(* revision histroy
hm	18. jun. 2008	rev 1.0
	original release

hm	20. sep. 2008	rev 1.1
	changed length of input string from 20 to 12
*)	
END_FUNCTION

(* POU String/BIN_TO_BYTE, ST *)
FUNCTION BIN_TO_BYTE : BYTE
VAR_INPUT
	BIN : STRING(12);
END_VAR
VAR
	pt : POINTER TO BYTE;
	i: INT;
	X: BYTE;
	stop: INT;
END_VAR

(*
version 1.1	20. sep. 2008
programmer 	hugo
tested by	oscat

BINARY_TO_byte converts a binary string into a byte.

*)
pt := ADR(bin);
stop := LEN(bin);
FOR I := 1 TO stop DO
	(* read the first character and subtract 48 to get value in decimal 0 = 48 *)
	x := pt^;
	(* calculate the value of the digit *)
	IF X = 48 OR X = 49 THEN
		BIN_TO_BYTE := SHL(BIN_TO_BYTE,1) + X - 48;
	END_IF;
	pt := pt + 1;
END_FOR;



(* revision histroy
hm	18. jun. 2008	rev 1.0
	original release

hm	20. sep. 2008	rev 1.1
	changed length of input string from 20 to 12

*)	
END_FUNCTION

(* POU String/OCT_TO_BYTE, ST *)
FUNCTION OCT_TO_BYTE : BYTE
VAR_INPUT
	OCT : STRING(10);
END_VAR
VAR
	pt : POINTER TO BYTE;
	i: INT;
	X: BYTE;
	stop: INT;
END_VAR

(*
version 1.1	20. sep. 2008
programmer 	hugo
tested by		oscat

OCT_TO_BYTE converts a octagonal string into a byte.

*)
pt := ADR(oct);
stop := LEN(oct);
FOR I := 1 TO stop DO
	(* read the first character and subtract 48 to get value in decimal 0 = 48 *)
	x := pt^;
	(* calculate the value of the digit *)
	IF X > 47 AND x < 56 THEN
		OCT_TO_BYTE := SHL(OCT_TO_BYTE,3) + X - 48;
	END_IF;
	pt := pt + 1;
END_FOR;



(* revision histroy
hm	18. jun. 2008	rev 1.0
	original release

hm	20. sep. 2008	rev 1.1
	changed length of input string from 20 to 10

*)	
END_FUNCTION

(* POU String/HEX_TO_BYTE, ST *)
FUNCTION HEX_TO_BYTE : BYTE
VAR_INPUT
	HEX : STRING(5);
END_VAR
VAR
	pt : POINTER TO BYTE;
	i: INT;
	X: BYTE;
	stop: INT;
END_VAR

(*
version 1.1	20. sep. 2008
programmer 	hugo
tested by		oscat

HEX_TO_BYTE converts a Hexadecimal string into a byte.

*)
pt := ADR(hex);
stop := LEN(hex);
FOR I := 1 TO stop DO
	(* read the first character and subtract 48 to get value in decimal 0 = 48 *)
	x := pt^;
	(* calculate the value of the digit *)
	IF X > 47 AND x < 58 THEN
		HEX_TO_BYTE := SHL(HEX_TO_BYTE,4) + X - 48;
	ELSIF X > 64 AND X < 71 THEN
		HEX_TO_BYTE := SHL(HEX_TO_BYTE,4) + X - 55;
	ELSIF X > 96 AND X < 103 THEN
		HEX_TO_BYTE := SHL(HEX_TO_BYTE,4) + X - 87;
	END_IF;
	pt := pt + 1;
END_FOR;




(* revision histroy
hm	18. jun. 2008	rev 1.0
	original release

hm	20. sep.2008	rev 1.1
	changed length of input string from 20 to 5

*)	
END_FUNCTION

(* POU String/DEC_TO_BYTE, ST *)
FUNCTION DEC_TO_BYTE : BYTE
VAR_INPUT
	DEC : STRING(10);
END_VAR
VAR
	pt : POINTER TO BYTE;
	i: INT;
	X: BYTE;
	stop: INT;
END_VAR

(*
version 1.1	30. sep 2008
programmer 	hugo
tested by		oscat

DEC_TO_byte converts a decimal string into a byte.

*)
pt := ADR(dec);
stop := LEN(DEC);
FOR I := 1 TO stop DO
	(* read the first character and subtract 48 to get value in decimal 0 = 48 *)
	x := pt^;
	(* calculate the value of the digit *)
	IF X > 47 AND x < 58 THEN
		DEC_TO_BYTE := DEC_TO_BYTE * 10 + X - 48;
	END_IF;
	pt := pt + 1;
END_FOR;



(* revision histroy
hm	20. jun. 2008	rev 1.0
	original release

hm	30. sep.2008	rev 1.1
	changed length of input string from 20 to 10
	corrected an error where decoding of characters 8 and 9 would fail

*)	
END_FUNCTION

(* POU String/CLEAN, ST *)
FUNCTION CLEAN : STRING(STRING_LENGTH)
VAR_INPUT
	IN : STRING(STRING_LENGTH);
	CX : STRING(80);
END_VAR
VAR
	pos: INT := 1;
	stop: INT;
END_VAR


(*
version 1.0	18. jun. 2008
programmer 	hugo
tested by	oscat

Clean deletes all characters from a string except the ones specified in CX.

*)
(* copy input string *)
CLEAN := IN;
stop := LEN(in);
WHILE pos <= stop DO
	IF FIND(cx, MID(CLEAN, 1, pos)) > 0 THEN
		(* charcter found skip to next one *)
		pos := pos + 1;
	ELSE
		(* wrong chracter needs to be deleted *)
		CLEAN := DELETE(CLEAN, 1, pos);
		stop := stop - 1;	(* the string is one character shorter now *)
	END_IF;
END_WHILE;



(* revision history

hm		18. jun. 2008	rev 1.0		
	original version 


*)
END_FUNCTION

(* POU String/IS_CC, ST *)
FUNCTION IS_CC : BOOL
VAR_INPUT
	str : STRING(STRING_LENGTH);
	cmp : STRING(STRING_LENGTH);
END_VAR
VAR
	L: INT;
	pos: INT;
END_VAR

(*
version 1.1	29. mar. 2008
programmer 	Tobias
tested by	hugo

ISC_CC testet ob ein string nur aus Zeichen des Strings CMP besteht.

*)
L := LEN(str);
FOR pos := 1 TO L DO
	IF FIND(CMP,MID(str,1,pos)) = 0 THEN RETURN; END_IF;
END_FOR;
IS_CC := L > 0;



(* revision history
hm	19. mar 2008	rev 1.0
	original version

hm	29. mar. 2008	rev 1.1
	changed STRING to STRING(STRING_LENGTH)
*)
END_FUNCTION

(* POU Mathematical/CMP, ST *)
FUNCTION CMP : BOOL
VAR_INPUT
	X,Y : REAL;
	N : INT;
END_VAR
VAR
	tmp : REAL;
END_VAR


(*
	version 1.0	12 mar 2008
	programmer 	hugo
	tested by		tobias

this function checks two inputs x and y if they are identical with the first N digits
example : cmp(3.141516,3.141517,6 is true.

*)
tmp := ABS(x);
IF tmp > 0 THEN
	tmp := EXP10(FLOOR(LOG(tmp))-N+1);
ELSE
	tmp := EXP10(tmp);
END_IF;
CMP := ABS(X - Y) < tmp;


(* revision history
hm	12. mar. 2008	rev 1.0
	original version

*)
END_FUNCTION

(* POU Mathematical/EXP10, ST *)
FUNCTION EXP10 : REAL
VAR_INPUT
	X : REAL;
END_VAR
VAR
END_VAR

(*
version 1.0	 2 dec 2007
programmer 	hugo
tested by		tobias

this function calculates the exponent to the basis 10
exp10(3) = 1000

*)
EXP10 := EXP(X * 2.30258509299405);

(* revision history
hm	2. dec 2007		rev 1.0
	original version

*)
END_FUNCTION

(* POU String/FSTRING_TO_WEEK, ST *)
FUNCTION FSTRING_TO_WEEK : BYTE
VAR_INPUT
	WEEK : STRING(60);
	LANG : INT;
END_VAR
VAR
	pos: INT;
END_VAR


(*
version 1.1	25. oct. 2008
programmer 	hugo
tested by	oscat

FSTRING_TO_WEEK converts a list of weekdays into a byte where each bit represents a day of the week.
bit 6 = mo, 0 = su;

*)
pos := FIND(WEEK, ',');
WHILE pos > 0 DO
	FSTRING_TO_WEEK := FSTRING_TO_WEEK OR SHR(BYTE#128, FSTRING_TO_WEEKDAY(MID(WEEK, pos - 1, 1), LANG));
	WEEK := RIGHT(WEEK, LEN(Week) - pos);
	pos := FIND(WEEK, ',');
END_WHILE;
FSTRING_TO_WEEK := (FSTRING_TO_WEEK OR SHR(BYTE#128, FSTRING_TO_WEEKDAY(WEEK, LANG))) AND BYTE#127;


(* revision histroy
hm	18. jun. 2008	rev 1.0
	original release

hm	25. oct. 2008	rev 1.1
	using language defauls and input lang
*)	
END_FUNCTION

(* POU String/FSTRING_TO_WEEKDAY, ST *)
FUNCTION FSTRING_TO_WEEKDAY : INT
VAR_INPUT
	WDAY : STRING(20);
	LANG : INT;
END_VAR
VAR
	tmp: STRING(2);
	i: INT;
	ly: INT;
END_VAR


(*
version 1.2	25. oct. 2008
programmer 	hugo
tested by	oscat

FSTRING_TO_WEEKDAY converts a weekday string into an integer 1..7.

*)
IF LANG = 0 THEN ly := LANGUAGE.DEFAULT; ELSE ly := MIN(LANG, LANGUAGE.LMAX); END_IF;
(* tmp needs to be calculated first otherwise find can return wrong values *)
tmp := TRIM(wday);
tmp := CAPITALIZE(LOWERCASE(tmp));
FOR i := 1 TO 7 DO
	IF language.WEEKDAYS2[ly, i] = tmp THEN
		FSTRING_TO_WEEKDAY := i;
		RETURN;
	END_IF;
END_FOR
FSTRING_TO_WEEKDAY := STRING_TO_INT(WDAY);




(* revision histroy
hm	18. jun. 2008	rev 1.0
	original release

hm	18. jul. 2008	rev 1.1
	changed nested call of left(trim()) for compatibility reasons

hm	25. oct. 2008	rev 1.2
	using language constants
*)	
END_FUNCTION

(* POU String/TRIM, ST *)
FUNCTION TRIM : STRING(STRING_LENGTH)
VAR_INPUT
	str : STRING(STRING_LENGTH);
END_VAR
VAR
	pos: INT;
END_VAR

(*
version 1.2	29. mar. 2008
programmer 	hugo
tested by	tobias

the function deletes all blanks within a string.

*)
TRIM := str;
REPEAT
	pos := FIND(trim,' ');
	IF pos > 0 THEN TRIM := REPLACE(TRIM,'',1,pos); END_IF;
UNTIL pos = 0	END_REPEAT;


(* revision histroy
hm	6.10.2006		rev 1.0
	original release

hm	20. mar. 2008	rev 1.1
	avoid to call replace with pos = 0 because some systems will produce an error

hm	29. mar. 2008	rev 1.2
	changed STRING to STRING(STRING_LENGTH)
*)
END_FUNCTION

(* POU String/CAPITALIZE, ST *)
FUNCTION CAPITALIZE : STRING(STRING_LENGTH)
VAR_INPUT
	str : STRING(STRING_LENGTH);
END_VAR
VAR
	PT : POINTER TO BYTE;
	pos : INT;
	L : INT;
	first : BOOL := TRUE;
END_VAR

(*
version 1.2	20. jun. 2008
programmer 	hugo
tested by		tobias

capitalize returns str with all first letters after a blank or beginning of the string are converted to uppercase.

*)
PT := ADR(CAPITALIZE);
CAPITALIZE := str;
L := LEN(str);
FOR pos := 1 TO l DO
	IF first THEN pt^ := TO_UPPER(pt^);	END_IF;
	(* remember in first if the next char needs to capitalized *)
	first := pt^= 32;
	PT := pt + 1;
END_FOR;

(* revision histroy
hm		4. mar 2008	rev 1.0
	original release

hm	29. mar. 2008	rev 1.1
	changed STRING to STRING(STRING_LENGTH)

hm	20. jun. 2008	rev 1.2
	improved performance

*)	
END_FUNCTION

(* POU String/TO_UPPER, ST *)
FUNCTION TO_UPPER : BYTE
VAR_INPUT
	IN : BYTE;
END_VAR
VAR
END_VAR

(*
version 1.3	16. jan. 2009
programmer 	hugo
tested by		oscat

to_upper converts a character from lowercase to uppercase

*)
IF in > 96 AND in < 123 THEN
   TO_UPPER := in AND 16#DF;
ELSIF in > 223 AND in <> 247 AND in <> 255 AND setup.EXTENDED_ASCII THEN
   TO_UPPER := in AND 16#DF;
ELSE
   TO_UPPER := in;
END_IF;




(* revision history
hm	6. mar. 2008	rev 1.0
	original version

hm	19. oct. 2008	rev 1.1
	changed setup constants

ks	25. oct. 2008	rev 1.2
	optimized code

hm 16. jan 2009	rev 1.3
	corrected an error in module

*)
END_FUNCTION

(* POU String/LOWERCASE, ST *)
FUNCTION LOWERCASE : STRING(STRING_LENGTH)
VAR_INPUT
	str : STRING(STRING_LENGTH);
END_VAR
VAR
	PT : POINTER TO BYTE;
	pos: INT;
	l: INT;
END_VAR

(*
version 1.3	29. mar. 2008
programmer 	hugo
tested by		tobias

lowercase returns str while all letters A..Z and Ä.Ö,Ü are converted to lowercase.

*)
PT := ADR(LOWERCASE);
lowercase := str;
l := LEN(str);
FOR pos := 1 TO l DO
	pt^ := TO_LOWER(pt^);
	PT := PT + 1;
END_FOR;

(* revision histroy
hm	6. oct. 2006	rev 1.0
	original release

hm	4. feb. 2008	rev 1.1
	improved performance
	added Ä.Ö,Ü

hm	6. mar. 2008	rev 1.2
	added support for exteded Ascii

hm	29. mar. 2008	rev 1.3
	changed STRING to STRING(STRING_LENGTH)
*)	
END_FUNCTION

(* POU String/TO_LOWER, ST *)
FUNCTION TO_LOWER : BYTE
VAR_INPUT
	IN : BYTE;
END_VAR
VAR
END_VAR

(*
version 1.2	25. oct 2008
programmer 	hugo
tested by		tobias

to_lower converts a character from uppercase to lowercase

*)
IF in > 64 AND in < 91 THEN
   TO_LOWER := in OR 16#20;
ELSIF (in > 191 AND in < 223) AND in <> 215 AND setup.EXTENDED_ASCII THEN
   TO_LOWER := in OR 16#20;
ELSE
   TO_LOWER := in;
END_IF;


(* revision history
hm	6. mar. 2008	rev 1.0
	original version

hm	19. oct. 2008	rev 1.1
	changed setup constants

ks	25. oct. 2008	rev 1.2
	optimized code
*)
END_FUNCTION

(* POU Building/electrical/TIMER_EXT, ST *)
FUNCTION_BLOCK TIMER_EXT
VAR_INPUT
	ENA : BOOL := TRUE;
	ON : BOOL;
	OFF : BOOL;
	MAN : BOOL;
	SWITCH : BOOL;
	DT_IN : DT;
	SUN_RISE : TOD;
	SUN_SET : TOD;
	HOLIDAY : BOOL;
END_VAR
VAR_INPUT CONSTANT
	T_DEBOUNCE : TIME := T#100ms;
	T_RISE_START : TIME;
	T_RISE_STOP : TIME;
	T_SET_START : TIME;
	T_SET_STOP : TIME;
	T_DAY_START : TOD;
	T_DAY_STOP : TOD;
	ENABLE_SATURDAY : BOOL;
	ENABLE_SUNDAY : BOOL;
	ENABLE_HOLIDAY : BOOL;
END_VAR
VAR_OUTPUT
	Q : BOOL;
	STATUS: BYTE;
END_VAR
VAR
	mx : MANUAL_2;
	deb : DEBOUNCE;
	tdx: TOD;
	wdx: INT;
	tc : TIME;
	tx: DWORD;
	tl: DWORD;
	qx: BOOL;
	init: BOOL;
END_VAR

(*
version 1.1	6. nov. 2008
programmer 	oscat
tested by	tobias

TIMER_EXT is a twilight timer.
the timer can be programmed to switch lights or other equippment or during twilight times.
in addition to the automatik mode the timer can be stopped and started by a switch at any given time.
An enable input ENA can be used for external control.
two inputs ON and OFF can be used to statically control the output.
the timer can be programmed to work on saturdays, sundays and holidays if required.

*)
(* lösche die millisekunden bei sunrise und sunset *)
SUN_RISE := DWORD_TO_TOD(TOD_TO_DWORD(SUN_RISE) / 1000 * 1000);
SUN_SET := DWORD_TO_TOD(TOD_TO_DWORD(SUN_SET) / 1000 * 1000);

(* measure cycle time tc and make sure this circuitry is not called more then once in 200ms*)
tx := T_PLC_MS();
IF NOT init THEN
	init := TRUE;
	tl := tx;
END_IF;
tc := DWORD_TO_TIME(tx - tl);
IF tc < t#200ms THEN RETURN; END_IF;
tl := tx;

(* debounce *)
deb(in := SWITCH, TD := T_DEBOUNCE, PM := TRUE);

(* read time of day and strip off all milliseconds *)
tdx := DT_TO_TOD(dt_in);
wdx := DAY_OF_WEEK(DT_TO_DATE(dt_in));

(* automatic output control *)
IF deb.Q THEN
	qx := NOT qx;
	status := 110;
ELSIF holiday AND NOT enable_holiday THEN
	qx := FALSE;
ELSIF wdx = 6 AND NOT enable_saturday THEN
	qx := FALSE;
ELSIF wdx = 7 AND NOT enable_sunday THEN
	qx := FALSE;
ELSIF T_day_start > TOD#00:00 AND tdx - T_DAY_START <= tc THEN
	(* turn on at specified daytime *)
	qx := TRUE;
	status := 111;
ELSIF T_DAY_STOP > TOD#00:00 AND tdx - T_DAY_STOP <= tc THEN
	(* turn off at specific daytime *)
	qx := FALSE;
	status := 112;
ELSIF T_RISE_START > T#0s AND tdx - SUN_RISE + T_RISE_START <= tc THEN
	(* turn on before sunrise *)
	qx := TRUE;
	status := 113;
ELSIF T_RISE_STOP > T#0s AND tdx - SUN_RISE - T_RISE_STOP <= tc THEN
	(* turn off after sunrise *)
	qx := FALSE;
	status := 114;
ELSIF T_SET_start > T#0s AND tdx - SUN_SET + T_SET_START <= tc THEN
	(* turn on before sunset *)
	qx := TRUE;
	status := 115;
ELSIF T_SET_STOP > t#0s AND tdx - SUN_SET - T_SET_STOP <= tc THEN
	(* turn off after sunset *)
	qx := FALSE;
	status := 116;
END_IF;


(* mnaual and output control *)
mx(in := qx, ena := ENA, on := ON, off := OFF, man := MAN);
Q := mx.Q;

(* set the status output *)
IF mx.STATUS > 100 THEN status := mx.STATUS; END_IF;



(*
hm 	7. oct. 2008	rev 1.0
	original version

hm	6. nov. 2008	rev 1.1
	added default = true for ena input
*)
END_FUNCTION_BLOCK

(* POU Engineering/automation/MANUAL_2, ST *)
FUNCTION_BLOCK MANUAL_2
VAR_INPUT
	IN : BOOL;
	ENA : BOOL;
	ON : BOOL;
	OFF : BOOL;
	MAN : BOOL;
END_VAR
VAR_OUTPUT
	Q : BOOL;
	STATUS : BYTE;
END_VAR
VAR
END_VAR

(*
version 1.0	22. sep. 2008
programmer 	hugo
tested by	oscat

MANUAL_2 is a manual override for boolean signals.
it has static force high and low as well as a manual input.

*)
IF ena THEN
	IF NOT ON AND NOT OFF THEN
		Q := IN;
		STATUS := 100;
	ELSIF on AND NOT off THEN
		Q := TRUE;
		STATUS := 101;
	ELSIF NOT on AND off THEN
		q := FALSE;
		STATUS := 102;
	ELSE
		Q := MAN;
		STATUS := 103;
	END_IF;
ELSE
	Q := FALSE;
	STATUS := 104;
END_IF;



(* revision history
hm	22. sep. 2008		rev 1.0
	original version

*)
END_FUNCTION_BLOCK

(* POU Building/electrical/TIMER_P4, ST *)
FUNCTION_BLOCK TIMER_P4
VAR_INPUT
	DTIME : DT;
	TREF_0 : TOD;
	TREF_1 : TOD;
	HOLY : BOOL;
	L0, L1, L2, L3 : BOOL;
	OFS : BYTE;
	ENQ : BOOL;
	MAN : BOOL;
	MI : BYTE;
	RST : BOOL;
END_VAR
VAR_IN_OUT
	PROG : ARRAY[0..array_max] OF TIMER_EVENT;
END_VAR
VAR_OUTPUT
	Q0, Q1, Q2, Q3 : BOOL;
	STATUS : BYTE;
END_VAR
VAR CONSTANT
	array_max : INT := 63;
	channel_max : INT := 3;
END_VAR
VAR
	event : TIMER_EVENT;
	pos : INT;
	last_execute: DT;
	current_day : DWORD;
	mask: BYTE;
	ma : ARRAY[0..channel_max] OF BYTE;
	mo : ARRAY[0..channel_max] OF BYTE;
	qn : ARRAY[0..channel_max] OF BOOL;
	channel: INT;
	tx: TOD;
END_VAR


(*
version 1.3	28. feb. 2009
programmer 	hugo
tested by		oscat

TIMER_P4 is a programmable universal timer.


*)
(* for performance reasons we only execute the code at the beginning of a new second
	we cannot compare the dtime directly because a daylight savings time switch might have happened
	therefore we need to compare the seconds and minutes of the dtime only 
	if we would compare seconds only the module would be in troulbe when its only called every minute 
	with this code the module is called every start of a new second *)

IF RST THEN
	last_execute := DT#1970-1-1-00:00;
	FOR pos := 0 TO ARRAY_MAX DO
		IF (PROG[pos].CHANNEL >= OFS) AND (PROG[pos].CHANNEL < (OFS + 4)) THEN PROG[pos].LAST := 0; END_IF;
	END_FOR;
ELSIF dtime <> last_execute THEN
	(* prepare the logical input mask to be used later *)
	mask := 255;
	mask.0 := L0;
	mask.1 := L1;
	mask.2 := L2;
	mask.3 := L3;
	(* save the actual second for next execution test *)
	last_execute := DTIME;
	current_day := DINT_TO_DWORD(DAY_OF_DATE(DT_TO_DATE(Dtime)));
	FOR pos := 0 TO ARRAY_MAX DO
		event := prog[pos];
		channel := event.CHANNEL - OFS;
		IF (event.TYP > 0) AND (channel >= 0) AND (channel <= channel_max) THEN
			ma[channel] := event.LAND;
			mo[channel] := event.LOR;
			CASE event.TYP OF
				1:	(* daily event *)
					qn[channel] := (DT_TO_TOD(dtime) >= event.START) AND (DT_TO_TOD(dtime) < event.START + event.DURATION);
					prog[pos].LAST := current_day;
				2: 	(* event by selected weekdays *)
					qn[channel] := (DT_TO_TOD(dtime) >= event.START) AND (DT_TO_TOD(dtime) < event.START + event.DURATION) AND ((SHR(BYTE#128, DAY_OF_WEEK(DT_TO_DATE(Dtime))) AND event.DAY) > 0);
					prog[pos].LAST := current_day;
				3:	(* event every N days *)
					qn[channel] := (DT_TO_TOD(dtime) >= event.START) AND (DT_TO_TOD(dtime) < event.START + event.DURATION) AND (event.LAST + event.DAY >= current_day);
					prog[pos].LAST := current_day;
				10:	(* weekly event exactly once a week the weekday is specified in day, 1= mo *)
					qn[channel] := (DT_TO_TOD(dtime) >= event.START) AND (DT_TO_TOD(dtime) < event.START + event.DURATION) AND DAY_OF_WEEK(DT_TO_DATE(DTIME)) = BYTE_TO_INT(event.DAY);
					prog[pos].LAST := current_day;
				20:	(* monthly event *)
					qn[channel] := (DT_TO_TOD(dtime) >= event.START) AND (DT_TO_TOD(dtime) < event.START + event.DURATION) AND DAY_OF_MONTH(DT_TO_DATE(DTIME)) = BYTE_TO_INT(event.DAY);
					prog[pos].LAST := current_day;
				21:	(* event on last day of month *)
					qn[channel] := (DT_TO_TOD(dtime) >= event.START) AND (DT_TO_TOD(dtime) < event.START + event.DURATION) AND (DT_TO_DATE(DTIME) = MONTH_END(DT_TO_DATE(dtime)));
					prog[pos].LAST := current_day;
				30:	(* yearly event on a specific day specified in day *)
					qn[channel] := (DT_TO_TOD(dtime) >= event.START) AND (DT_TO_TOD(dtime) < event.START + event.DURATION) AND DAY_OF_YEAR(DT_TO_DATE(DTIME)) = BYTE_TO_INT(event.DAY);
					prog[pos].LAST := current_day;
				31:	(* event on last day of year *)
					qn[channel] := (DT_TO_TOD(dtime) >= event.START) AND (DT_TO_TOD(dtime) < event.START + event.DURATION) AND (DT_TO_DATE(DTIME) = YEAR_END(YEAR_OF_DATE(DT_TO_DATE(dtime))));
					prog[pos].LAST := current_day;
				40:	(* event on leap days *)
					qn[channel] := (DT_TO_TOD(dtime) >= event.START) AND (DT_TO_TOD(dtime) < event.START + event.DURATION) AND LEAP_DAY(DT_TO_DATE(dtime));
					prog[pos].LAST := current_day;
				41: (* event on holidays *)
					qn[channel] := (DT_TO_TOD(dtime) >= event.START) AND (DT_TO_TOD(dtime) < event.START + event.DURATION) AND HOLY;
					prog[pos].LAST := current_day;
				42: (* event on holidays and weekends *)
					qn[channel] := (DT_TO_TOD(dtime) >= event.START) AND (DT_TO_TOD(dtime) < event.START + event.DURATION) AND (Holy OR (DAY_OF_WEEK(DT_TO_DATE(dtime)) = 6) OR (DAY_OF_WEEK(DT_TO_DATE(dtime)) = 7));
					prog[pos].LAST := current_day;
				43:	(* event on workdays Mo-FR and no holiday *)
					qn[channel] := (DT_TO_TOD(dtime) >= event.START) AND (DT_TO_TOD(dtime) < event.START + event.DURATION) AND (NOT Holy) AND (DAY_OF_WEEK(DT_TO_DATE(dtime)) < 6);
					prog[pos].LAST := current_day;
				50: (* event after reference time *)
					CASE prog[pos].DAY OF
						0:	tx := tref_0;
						1:	tx := tref_1;
					ELSE
						tx := TOD#00:00;
					END_CASE;
					qn[channel] := (DT_TO_TOD(dtime) >= (tx + TOD_TO_TIME(event.START))) AND (DT_TO_TOD(dtime) < (tx + TOD_TO_TIME(event.START) + event.duration));
					prog[pos].LAST := current_day;
				51:	(* event before reference time *)
					CASE prog[pos].DAY OF
						0:	tx := tref_0;
						1:	tx := tref_1;
					ELSE
						tx := TOD#00:00;
					END_CASE;
					qn[channel] := (DT_TO_TOD(dtime) >= (tx - TOD_TO_TIME(event.START))) AND (DT_TO_TOD(dtime) < (tx - TOD_TO_TIME(event.START) + event.duration));
					prog[pos].LAST := current_day;
				52 : (* enable output at specific time + offset  *)
					CASE prog[pos].DAY OF
						0:	tx := tref_0;
						1:	tx := tref_1;
					ELSE
						tx := TOD#00:00;
					END_CASE;
					IF (DT_TO_TOD(dtime) >= tx + TOD_TO_TIME(event.START)) AND (event.LAST <> current_day) THEN
						qn[channel] := TRUE;
						prog[pos].LAST := current_day;
					END_IF;
				53 : (* disable output at specific time + offset *)
					CASE prog[pos].DAY OF
						0:	tx := tref_0;
						1:	tx := tref_1;
					ELSE
						tx := TOD#00:00;
					END_CASE;
					IF (DT_TO_TOD(dtime) >= tx + TOD_TO_TIME(event.START)) AND (event.LAST <> current_day) THEN
						qn[channel] := FALSE;
						prog[pos].LAST := current_day;
					END_IF;
				54 : (* enable output at specific time - offset  *)
					CASE prog[pos].DAY OF
						0:	tx := tref_0;
						1:	tx := tref_1;
					ELSE
						tx := TOD#00:00;
					END_CASE;
					IF (DT_TO_TOD(dtime) >= tx - TOD_TO_TIME(event.START)) AND (event.LAST <> current_day) THEN
						qn[channel] := TRUE;
						prog[pos].LAST := current_day;
					END_IF;
				55 : (* disable output at specific time - offset *)
					CASE prog[pos].DAY OF
						0:	tx := tref_0;
						1:	tx := tref_1;
					ELSE
						tx := TOD#00:00;
					END_CASE;
					IF (DT_TO_TOD(dtime) >= tx - TOD_TO_TIME(event.START)) AND (event.LAST <> current_day) THEN
						qn[channel] := FALSE;
						prog[pos].LAST := current_day;
					END_IF;
			END_CASE;
		END_IF;
	END_FOR;
END_IF;

(* set the outputs *)
Q0 := ENQ AND (qn[0] AND ((ma[0] AND mask) = ma[0]) OR ((mo[0] AND mask) > 0) OR (man AND MI.0));
Q1 := ENQ AND (qn[1] AND ((ma[1] AND mask) = ma[1]) OR ((mo[1] AND mask) > 1) OR (man AND MI.1));
Q2 := ENQ AND (qn[2] AND ((ma[2] AND mask) = ma[2]) OR ((mo[2] AND mask) > 2) OR (man AND MI.2));
Q3 := ENQ AND (qn[3] AND ((ma[3] AND mask) = ma[3]) OR ((mo[3] AND mask) > 3) OR (man AND MI.3));

(* set status *)
IF NOT enq THEN
	status := 100;
ELSIF man THEN
	status := 101;
ELSE
	status := 102;
END_IF;




(* revision history
hm	17. jun 2008	rev 1.0
	original version

hm	9. oct. 2008	rev 1.1
	changed function year to year_of_date
	changed function weekday to day_of_week
	changed structure of program to be more efficient
	changed input DIS to ENQ

hm	18. oct. 2008	rev 1.2
	changed type of input OFS from int to byte
	added typecasts to avoid warnings

hm	28. feb. 2009	rev 1.3
	array was not correctly initialized

*)
END_FUNCTION_BLOCK

(* POU Mathematical/Array/ARRAY_MAX, ST *)
FUNCTION ARRAY_MAX : REAL
VAR_INPUT
	pt : POINTER TO ARRAY[0..32000] OF REAL;
	size : UINT;
END_VAR
VAR
	i: UINT;
	stop: UINT;
END_VAR

(*
version 1.1	16. mar. 2008
programmer 	hugo
tested by		tobias

this function will calculate the max value of a given array.
the function needs to be called:	array_max(adr("array"),sizeof("array"));
because this function works with pointers its very time efficient and it needs no extra memory.

*)
stop := (size -SIZEOF(pt)) / SIZEOF(pt);
array_max := pt^[0];
FOR i := 1 TO stop DO
	IF pt^[i] > array_max THEN array_max := pt^[i]; END_IF;
END_FOR;

(* revision history
hm	2. oct 2006		rev 1.0
	original version

hm	16. mar. 2008	rev 1.1
	changed input size to uint
*)
END_FUNCTION

(* POU Time&Date/DAY_OF_DATE, ST *)
FUNCTION DAY_OF_DATE : DINT
VAR_INPUT
	idate : DATE;
END_VAR
VAR
END_VAR


(*
	version 1.3	7. apr. 2008
	programmer 	oscat
	tested BY	oscat

DAY_OF_DATE returns the days since 1.1.1970

*)
DAY_OF_DATE := DWORD_TO_DINT(DATE_TO_DWORD(idate) / 86400);


(* revision history
hm		16.9.2007		rev 1.0
	original version

hm		1. okt 2007		rev 1.1
	added step7 compatibility

hm		22. mar. 2008	rev 1.2
	changed output from int to Dint because the total date range is 49710 days

hm		7. apr. 2008	rev 1.3
	deleted unused step7 code

*)
END_FUNCTION

(* POU Time&Date/MONTH_END, ST *)
FUNCTION MONTH_END : DATE
VAR_INPUT
	IDATE : DATE;
END_VAR
VAR
END_VAR

(*
version 1.1	7. oct. 2008
programmer 	hugo
tested by	oscat

returns the date for the last day of the current month in the current year.

*)
MONTH_END := DWORD_TO_DATE(DATE_TO_DWORD(SET_DATE(YEAR_OF_DATE(idate),MONTH_OF_DATE(idate)+1,1)) - 86400);



(* revision history
hm	15. jun. 2008	rev 1.0
	original version	

hm	7. oct. 2008	rev 1.1
	changed function year to year_of_date
	changed function month to month_of_date

*)
END_FUNCTION

(* POU Time&Date/YEAR_END, ST *)
FUNCTION YEAR_END : DATE
VAR_INPUT
	y : INT;
END_VAR
VAR
END_VAR

(*
version 1.0	15. jun. 2008
programmer 	hugo
tested by	oscat

returs the date of december 31st for the given year  
the function works for dates from 1970 - 2099 

*)
YEAR_END := DWORD_TO_DATE(SHR(INT_TO_DWORD(y+1) * 1461 - 2878173,2)*86400);



(* revision history
hm	15. jun. 2008	rev 1.0
	original version

*)
END_FUNCTION

(* POU Time&Date/LEAP_DAY, ST *)
FUNCTION LEAP_DAY : BOOL
VAR_INPUT
	IDATE : DATE;
END_VAR
VAR
END_VAR

(*
version 1.1	7. oct. 2008
programmer 	hugo
tested by	oscat


leap_day is true if the tested day is a leap day (29. of february).  
  
*)
LEAP_DAY := (MONTH_OF_DATE(idate) = 2) AND (DAY_OF_MONTH(idate) = 29);



(* change history

hm 	15. jun. 2008	rev 1.0
	original version

hm	7. oct. 2008	rev 1.1
	changed function month to month_of_date
*)
END_FUNCTION

(* POU Building/HLK/AIR_DENSITY, ST *)
FUNCTION AIR_DENSITY : REAL
VAR_INPUT
	T : REAL;
	P : REAL;
	RH : REAL;
END_VAR
VAR CONSTANT
	RL : REAL := 287.05;
	RX : REAL := 3.773319E-3;
END_VAR
VAR
END_VAR

(*
version 1.2	18. oct. 2008
programmer 	hugo
tested by		tobias

this function calculates the air density between 0 and 100 deg C

*)
AIR_DENSITY := phys.PN * (1 - RH * SDD(T, TRUE) * RX / P) / (RL * ( T - phys.T0));

(* original code used for rev 1.0

SDD := SDD(T,FALSE);
RF := RL / (1- RH*SDD/P*RX);
Air_density := P / (RF * (T-TK));

*)

(* revision history

hm	29.10.2007		rev 1.0
	original version

hm	4.12.2007		rev 1.1
	changed code for better performance

hm	18. oct. 2008	rev 1.2
	using phys constants

*)
END_FUNCTION

(* POU Building/HLK/SDD, ST *)
FUNCTION SDD : REAL
VAR_INPUT
	T : REAL;
	ICE: BOOL;
END_VAR
VAR CONSTANT
END_VAR
VAR
END_VAR

(*
version 1.1	2 dec 2007
programmer 	hugo
tested by		tobias

this function calculates the vapor saturation pressure for moist Air over ice or water

*)
IF ice THEN
	SDD := 611.153 * EXP(22.4433 * T / (272.186 + T));
ELSE
	SDD := 611.213 * EXP(17.5043 * T / (241.2 + T));
END_IF;

(* old code used in rev 1.0
IF ice THEN
	SDD := 611.153 * exp10(9.747*T / (272.186 + T));
ELSE
	SDD := 611.213 * exp10(7.602*T / (241.2 + T));
END_IF;
*)


(* revision history

hm 29 oct 2007		rev 1.0
	original version

hm	2. dec 2007		rev 1.1
	changed code for better performance
*)
END_FUNCTION

(* POU Building/HLK/AIR_ENTHALPY, ST *)
FUNCTION AIR_ENTHALPY : REAL
VAR_INPUT
	T : REAL;
	RH : REAL;
END_VAR
VAR CONSTANT
	CPL : REAL := 1.00482;
	CW : REAL := 1.86;
	LH : REAL := 2500.78;
END_VAR
VAR
END_VAR

(*
version 1.1	2 nov 2007
programmer 	hugo
tested by		tobias

this function calculates the enthalpy for humid air between 0 and 100 deg C

*)
Air_enthalpy := CPL * T + (CW * T + LH) * dew_con(RH,T);

(* revision history

hm	31.10.2007		rev 1.0
	original version

hm	2.11.2007		rev 1.1
	deleted unused variable RF

hm	2.12.2007		rev 1.2
	changed code for better performance
*)
END_FUNCTION

(* POU Building/HLK/DEW_CON, ST *)
FUNCTION DEW_CON : REAL
VAR_INPUT
	RH : REAL;
	T : REAL;
END_VAR
VAR CONSTANT
END_VAR
VAR
END_VAR

(*
version 1.4	18. oct. 2008
programmer 	hugo
tested by	oscat

this function calculates the water concentratin in air for a given temperature and relative humidity.
the output states the concentration of water vapor in air in Gramms / qubic meter.

*)
(*	this code is good to read but need to be improoved
	SDD := 6.1078*EXPT(10,(a*T)/(b+T));
	DD := RH/100 * SDD;
	V := LOG(DD/6.1078);
	TD := b*V/(a-v);
	dew_con := 0.1 * mw / RU * DD / (T - TK);
*)
DEW_CON := 2.166824303E-2 * RH * SDD(T,FALSE)  / (T - phys.T0) * BOOL_TO_INT(RH > 0);


(*
Bezeichnungen:
r = relative Luftfeuchte
T = Temperatur in °C
TK = Temperatur in Kelvin (TK = T + 273.15)
TD = Taupunkttemperatur in °C
DD = Dampfdruck in hPa
SDD = Sättigungsdampfdruck in hPa

Parameter:
a = 7.5, b = 237.3 für T >= 0
a = 7.6, b = 240.7 für T < 0 über Wasser (Taupunkt)
a = 9.5, b = 265.5 für T < 0 über Eis (Frostpunkt)

R* = 8314.3 J/(kmol*K) (universelle Gaskonstante)
mw = 18.016 kg (Molekulargewicht des Wasserdampfes)
AF = absolute Feuchte in g Wasserdampf pro m3 Luft

Formeln:

   1. SDD(T) = 6.1078 * 10^((a*T)/(b+T))
   2. DD(r,T) = r/100 * SDD(T)
   3. r(T,TD) = 100 * SDD(TD) / SDD(T)
   4. TD(r,T) = b*v/(a-v) mit v(r,T) = log10(DD(r,T)/6.1078)
   5. AF(r,TK) = 10^5 * mw/R* * DD(r,T)/TK; AF(TD,TK) = 10^5 * mw/R* * SDD(TD)/TK 

*)

(* revision history

hm 29 apr 2007		rev 1.0
	original version

hm	13.sep 2007		rev 1.1
	improoved coding for speed
	deleted unused variabled SDD,DD,V, TD

hm	2. dec 2007		rev 1.2
	changed code for better performance
	output is now in Gramms / Qubic meter

hm	14. oct. 2008	rev 1.3
	performance improvement

hm	18. oct. 2008	rev 1.4
	using phys constants

*)
END_FUNCTION

(* POU Building/HLK/BOILER, ST *)
FUNCTION_BLOCK BOILER
VAR_INPUT
	T_upper : REAL;
	T_lower : REAL;
	Pressure : BOOL := TRUE;
	enable : BOOL := TRUE;
	Req_1 : BOOL;
	Req_2 : BOOL;
	Boost : BOOL;
END_VAR
VAR_INPUT CONSTANT
	t_upper_min : REAL := 50;
	t_upper_max : REAL := 60;
	T_lower_enable : BOOL;
	T_lower_max : REAL := 60;
	T_request_1 : REAL := 70;
	T_request_2 : REAL := 50;
	T_request_hys : REAL := 5;
	T_protect_high : REAL := 80;
	T_protect_low : REAL := 10;
END_VAR
VAR_OUTPUT
	Heat : BOOL;
	error : BOOL;
	status : BYTE;
END_VAR
VAR
	edge: BOOL;
	boost_mode: BOOL;
	flag_0 : BOOL;
	flag_1: BOOL;
	flag_2: BOOL;
END_VAR

(*
version 1.1	16. oct. 2008
programmer 	hugo
tested by	oscat


this function block controls a hot water boiler. The Boiler can be equipped with two temperature sensors on top and bottom of the tank, T_LOWER_ENABLE must be set to True in this case.
alternatively can BOILER be configured for one (TOP) temperature sensor only (T_LOWER_ENABLE set to False).
A Pressure sensor is used to detect fresh water pressure and disable all heating if there is no water pressure. This input is dset to True by default, so if it is not used it can simply be left open.
A enable input enables the hot water heating while it is set to True. alternatively can a Ture on Req_1 or Req_2 start the heating to predefined temperatures during setup.
A low to high edge on the boost input will start heating imediately until T_upper_max is reached, it can be used to generate extra hot water when needed.

*)
(* read sensors and check for valid data *)
IF t_upper > t_protect_high THEN
	status := 1;
	heat := FALSE;
	error := TRUE;
ELSIF t_upper < t_protect_low THEN
	status := 2;
	heat := error := TRUE;
ELSIF t_lower > T_protect_high AND t_lower_enable THEN
	status := 3;
	heat := FALSE;
	error := TRUE;
ELSIF t_lower < t_protect_low AND t_lower_enable THEN
	status := 4;
	heat := error := TRUE;
ELSIF NOT pressure THEN
	status := 5;
	heat := FALSE;
	error := TRUE;
ELSIF req_1 OR req_2 OR enable OR boost THEN
	error := FALSE;

	(* determine if heat needs to be turned on *)
	IF boost AND NOT edge AND t_upper < t_upper_max THEN
		status := 101;
		heat := TRUE;
		boost_mode := TRUE;
	ELSIF enable AND t_upper < T_upper_min THEN
		status := 102;
		heat := TRUE;
	ELSIF req_1 AND t_upper < T_request_1 THEN
		status := 103;
		heat := TRUE;
	ELSIF req_2 AND t_upper < t_request_2 THEN
		status := 104;
		heat := TRUE;
	END_IF;

	(* determine the shut off temperature *)
	IF heat THEN
		IF (enable OR boost_mode) THEN
			flag_0 := TRUE;
			IF T_lower_enable AND T_lower > T_lower_max THEN
				flag_0 := boost_mode := FALSE;
			ELSIF NOT T_lower_enable AND T_upper > T_upper_max THEN
				flag_0 := boost_mode := FALSE;
			END_IF;
		ELSE
			flag_0 := FALSE;
		END_IF;
		flag_1 := (req_1 AND T_upper > T_request_1 + T_request_hys) AND req_1;
		flag_2 := (req_2 AND T_upper > T_request_2 + T_request_hys) AND req_2;

		(* shut off heat if no longer needed *)
		heat := flag_0 OR flag_1 OR flag_2;
		IF heat = FALSE THEN status := 100; END_IF;
	END_IF;
ELSE
	status := 100;
	heat := error := FALSE;
END_IF;
edge := boost;


(* revision history
hm	27. feb. 2007	rev 1.0
	original version

hm	16. oct. 2008	rev 1.1
	improved performance


*)
END_FUNCTION_BLOCK

(* POU Engineering/conversion/PRESSURE, ST *)
FUNCTION_BLOCK PRESSURE
VAR_INPUT
	mws : REAL;
	torr : REAL;
	att : REAL;
	atm : REAL;
	pa : REAL;
	bar : REAL;
END_VAR
VAR_OUTPUT
	Ymws : REAL;
	Ytorr : REAL;
	Yatt : REAL;
	Yatm : REAL;
	Ypa : REAL;
	Ybar : REAL;
END_VAR
VAR
END_VAR

(*
version 1.0	27 mar 2007
programmer 	hugo
tested by		oscat

this function converts different pressure units
any unused input can simply be left open.
different inputs connected at the same time will be added up.
*)
Ybar := bar +
		pa / 100000 +
		0.980665 * att +
		1.01325 * atm +
		0.001333224 * torr +
		0.0980665 * mws;
Ymws := ybar / 0.0980665;
Ytorr := ybar / 0.001333224;
Yatt := ybar / 0.980665;
yatm := ybar / 1.01325;
Ypa := ybar * 100000;


(*
Druck, Pascal Pa 1 Pa = 1 N/m2 = 1 kg/(s2 �E m) . 0,75 �E 10.2 mmHg
mechanische 1 MPa = 1 N/mm2 . fur Festigkeitsangaben
Spannung Bar bar 1 bar = 105 Pa = 103 mbar = 105 kg/(s2 �E m)
Millimeter- mmHg 1 mmHg = 133,322 Pa = 1,333 22 mbar
Quecksilbersaule . nur in Heilkunde zulassig
physik. Atmosphare atm 1 atm = 1,013 25 bar
techn. Atmosphare at 1 at = 1 kp/cm2 = 0,980665 bar
Torr Torr 1 Torr = (101325/760) Pa = 1,333224 mbar
Meter-Wassersaule mWS 1 mWS = 9806,65 Pa = 98,0665 mbar
psi lbf/in2 1 lbf/in2 = 68,947 57 mbar = 6894,757 Pa

*)
END_FUNCTION_BLOCK

(* POU Building/HLK/BURNER, ST *)
FUNCTION_BLOCK BURNER
VAR_INPUT
	in : BOOL;
	stage2 : BOOL;
	over_temp : BOOL;
	oil_temp : BOOL := TRUE;
	Flame : BOOL;
	rst : BOOL;
	rst_timer : BOOL;
END_VAR
VAR_INPUT CONSTANT
	pre_heat_time : TIME := t#5s;
	pre_vent_time : TIME := t#15s;
	pre_ignite_time : TIME := t#5s;
	post_ignite_time : TIME := t#25s;
	stage2_delay : TIME := t#10s;
	safety_time : TIME := t#5s;
	lockout_time : TIME := t#10s;
	multiple_ignition : BOOL := TRUE;
	KW1 : REAL;
	KW2 : REAL;
END_VAR
VAR_OUTPUT
	motor : BOOL;
	coil1 : BOOL;
	coil2 : BOOL;
	pre_heat: BOOL;
	ignite : BOOL;
	KWh : REAL;
	status : BYTE;
	fail : BOOL;
END_VAR
VAR_IN_OUT
	runtime1 : UDINT;
	runtime2 : UDINT;
	cycles : UDINT;
END_VAR
VAR
	state : BYTE;
	last : TIME;
	tx: TIME;
	last_change: TIME;
	timer1 : ONTIME;
	timer2 : ONTIME;
	oil_temp_last: BOOL;
	cycles2 : UDINT;
END_VAR

(*
version 1.5	15 sep 2007
programmer 	oscat
tested by	oscat

burner ist eine Oel-Brenner_steuerung fuer nichtmodulierende Oelbrenner
die steuerung kann ueber setup werte programmiert werden und entsprechenden brennern angepasst werden.
die vorheizzeit ist die zeit die eine oelvorwaermung aufgeheizt wird bevor der motor gestartet wird.
der eingang oil_temp gibt an ob die oil_temp erreicht wurde, er ist default auf true und kann auch offen gelassen werden.
die vorbelueftungszeit ist die zeit die der luefter laeuft bevor die oelzufuhr freigegeben wird.
die vorzuendzeit iust diejenige zeit die die zuendung vor offnen des oelventiel gestartet wird.
nachzuendzeit ist die zeit die nach entzuendung der flamme noch gezuendet wird.
die sicherheitszeit ist die zeit nach der die oelzufuhr gesperrt wird wenn keine flamme entsteht.
nach ablauf der sicherheitszeit wird ein fehler flag gesetzt und kann erst nach der sperrzeit wieder durch einen reset geloescht werden.
waehrend der sperrzeit ist keine weitere zuendung oder einschalten moeglich.
das flag mehrfachzuendung gibt an ob eine erloschene flamme in betrieb automatisch wieder gezuendet werden soll.
der flammwaechster liegt auf eingang flamme, ein uebertemperaturschutz auf dem eingang over_temp
der betriebsstundenzaehler gibt die brennerstunden in stunden als real ausgabewer an.
der ausgang motor steuert den luefter / pumpenmotor, oil_ventil schaltet das oil ventil und zuendung schaltet die zuendung ein.

if output fail > 0 an error happened and the output has an error code:
0 :	no error
1 :	pre heating time expired and oil temp input is not true
2 :	flame monitor is active during preheating time
3 :	flame monitor active during pre_ventilation_time
4 :	no ignoition during safety time
5 :	no flame during operation
9 :	overtemp input is true

*)
(* read system time *)
tx := DWORD_TO_TIME(T_PLC_MS());

(* check rst input and overtemp *)
IF rst OR over_temp OR state = 0 THEN
	IF status > 0 AND tx - last_change >= lockout_time AND rst THEN
		status := 110;
		fail := FALSE;
		state := 1;
	ELSE
		(* normaler reset *)
		motor := FALSE;
		coil1 := FALSE;
		coil2 := FALSE;
		ignite := FALSE;
		pre_heat := FALSE;
		IF over_temp THEN
			status := 9;
			fail := TRUE;
		END_IF;
		last_change := tx;
		last := tx;
		state := 1;
	END_IF;
END_IF;

(* check for timer rst and rst timer if true *)
IF rst_timer THEN
	runtime1 := 0;
	runtime2 := 0;
	cycles := 0;
	cycles2 := 0;
END_IF;

(* quit here if an error is present *)
IF (status > 0 AND status < 100) OR rst THEN RETURN; END_IF;

(* start sequence *)
CASE state OF

1:	(* in signal starts oil pre heating *)
	IF in AND flame THEN
		state := 7;
		pre_heat := FALSE;
		status := 2;
		last_change := tx;
	ELSIF in THEN
		pre_heat := TRUE;
		state := 2;
		last_change := tx;
	END_IF;

2:	(* after pre_heating time start motor *)
	IF (tx- last_change >= pre_heat_time AND oil_temp) OR (oil_temp AND NOT oil_temp_last) THEN
		motor := TRUE;
		state := 3;
		last_change := tx;
	(* pre_heat_time ist abgelaufen und oil_temp ist nicht aktiv *)
	ELSIF tx - last_change >= pre_heat_time AND NOT oil_temp THEN
		state := 7;
		pre_heat := FALSE;
		status := 1;
		last_change := tx;
	(* flame monitor cannot be active at this time *)
	ELSIF flame THEN
		state := 7;
		pre_heat := FALSE;
		status := 2;
		last_change := tx;
	END_IF;

3:	(* abwarten bis zündung eingeschaltet werden kann *)
	IF tx - last_change >= pre_vent_time - pre_ignite_time THEN
		ignite := TRUE;
		state := 4;
		last_change := tx;
	(* flame monitor cannot be active at this time *)
	ELSIF flame THEN
		state := 7;
		pre_heat := FALSE;
		motor := FALSE;
		status := 3;
		last_change := tx;
	END_IF;

4:	(* warten bis oelzufuhr geoeffnet werden darf *)
	IF tx - last_change >= pre_ignite_time THEN
		coil1 := TRUE;
		state := 5;
		last_change := tx;
	END_IF;

5:	(* warten auf flammwaechter und falls noetig abschalten *)
	IF tx - last_change >= safety_time OR flame THEN
		IF NOT flame THEN
			(* notabschaltung da flammwaechster nicht angesprochen hat *)
			state := 7;
			motor := FALSE;
			coil1 := FALSE;
			pre_heat := FALSE;
			ignite := FALSE;
			status := 4;
			last_change := tx;
		ELSE
			state := 6;
			last_change := tx;
		END_IF;
	END_IF;

6:	(* brenner läuft, flammueberwachung und nach ablauf der nachigniteszeit ignite abschalten *)
	IF NOT flame AND NOT multiple_ignition THEN
		(* notabschaltung da flammwaechster keine flamme meldet *)
		state := 7;
		motor := FALSE;
		coil1 := FALSE;
		coil2 := FALSE;
		pre_heat := FALSE;
		ignite := FALSE;
		status := 5;
		last_change := tx;
	ELSIF NOT flame AND multiple_ignition THEN
		ignite := TRUE;
		state := 5;
		coil2 := FALSE;
		last_change := tx;
	ELSE
		IF tx - last_change >= post_ignite_time THEN
			(* post_ignite_time abgelaufen, ignite abschalten *)
			ignite := FALSE;
		END_IF;
		IF tx - last_change >= stage2_delay AND stage2 THEN
			coil2 := TRUE;
		ELSE
			coil2 := FALSE;
		END_IF;
	END_IF;
END_CASE;

(* abschaltung wenn kein eingangssignal *)
IF NOT in THEN
	state := 1;
	motor := FALSE;
	coil1 := FALSE;
	coil2 := FALSE;
	ignite := FALSE;
	pre_heat := FALSE;
	last_change := tx;
END_IF;

(* runtimezähler *)
timer1(in := flame AND in AND motor AND coil1 AND NOT coil2, seconds := runtime1, cycles := cycles);
timer2(in := flame AND in AND motor AND coil1 AND coil2, seconds := runtime2, cycles := cycles2);
KWH := UDINT_TO_REAL(runtime1) * KW1 / 3600.0 + UDINT_TO_REAL(runtime2) * KW2 / 3600.0;

(* zeit fuer naechsten aufruf merken *)
last := tx;

(* set fail output IF ERROR and Status  if normal operation *)

IF status > 0 AND status < 100 THEN
	fail := TRUE;
ELSE
	fail := FALSE;
	IF NOT in THEN
		status := 110;
	ELSIF flame AND in AND motor AND coil2 AND coil1 THEN
		status := 113;
	ELSIF flame AND in AND motor AND coil1 THEN
		status := 112;
	ELSE
		status := 111;
	END_IF;
END_IF;



(*
31.12.2006	hm		rev 1.1
	added pre_heat timing and output
	flame monitor before ignition will generate error on status output
	added output for KWh

31.12.2006	hm		rev 1.2
	added oil_temp_input

31.12.2006	hm		rev 1.3
	changed status output to be byte instead of bool

22.1.2007		hm		rev 1.4
	renamed fail output to status
	added output cycles
	corrected an error while pre_heat would be on when an error was present
	added coil2 output and stage2 input

15.9.2007		hm		rev 1.5
	replaced Time() with T_PLC_MS for compatibility and performance reasons

hm	21. oct. 2008	rev 1.6
	changed code to use new ontime rev 2.0	
*)
END_FUNCTION_BLOCK

(* POU Building/HLK/DEW_RH, ST *)
FUNCTION DEW_RH : REAL
VAR_INPUT
	VC : REAL;
	T : REAL;
END_VAR

(*
version 1.1	2 dec 2007
programmer 	hugo
tested by		tobias

this function calculates the relative humidity in air for a given temperature in °C and vapor concentration in Kg/m³..

*)
dew_rh := LIMIT(0,VC / dew_con(1,T),100);

(* code before rev 1.1
dew_rh := VC / dew_con(100,T) * 100;
IF dew_rh > 100 THEN dew_rh := 100; END_IF;
*)

(* revision history
hm		29. apr 2007	rev 1.0
	original version

hm		2. 12. 2007		rev 1.1
	new code for better performance

*)
END_FUNCTION

(* POU Building/HLK/DEW_TEMP, ST *)
FUNCTION DEW_TEMP : REAL
VAR_INPUT
	RH : REAL;
	T : REAL;
END_VAR
VAR CONSTANT
	a : REAL := 7.5;
	b : REAL := 237.3;
END_VAR
VAR
	V : REAL;
END_VAR

(*
version 1.5	18. oct. 2008
programmer 	hugo
tested by	oscat

this function calculates the dew point for air given the temperature and relative humidity.
dew_temp(60,0.25) = 16.7 °C.
which means the dew point for air with 25° and 60% RH is at 16.7 °C.


*)
IF rh > 0 THEN
(*	old code was rewritten for better performance
	SDD := 6.1078*EXPT(10,(a*T)/(b+T));
	DD := RH/100 * SDD;
	V := LOG(DD/6.1078);
	dew_temp := b*V/(a-v);
*)
	V := LOG(RH * 0.01 * exp10((a*T)/(b+T)));
	dew_temp := b*V/(a-V);
ELSE
	DEW_TEMP:= - phys.T0;
END_IF;

(* revision history

hm		2.10.2006	rev 1.0
	original version created

hm		29.4.2007	rev 1.1
	checked for rh not to be 0 because log(0) is not defined

hm		13.9.2007	rev 1.2
	code rewritten for better performance

hm		2. dec 2007	rev 1.3
	changed code for better performance

hm		8. jan 2008	rev 1.4
	further improvement in performance

hm	18. oct. 2008	rev 1.5
	using phys constants	

*)

(*
Bezeichnungen:
r = relative Luftfeuchte
T = Temperatur in °C
TK = Temperatur in Kelvin (TK = T + 273.15)
TD = Taupunkttemperatur in °C
DD = Dampfdruck in hPa
SDD = Sättigungsdampfdruck in hPa

Parameter:
a = 7.5, b = 237.3 für T >= 0
a = 7.6, b = 240.7 für T < 0 über Wasser (Taupunkt)
a = 9.5, b = 265.5 für T < 0 über Eis (Frostpunkt)

R* = 8314.3 J/(kmol*K) (universelle Gaskonstante)
mw = 18.016 kg (Molekulargewicht des Wasserdampfes)
AF = absolute Feuchte in g Wasserdampf pro m3 Luft

Formeln:

   1. SDD(T) = 6.1078 * 10^((a*T)/(b+T))
   2. DD(r,T) = r/100 * SDD(T)
   3. r(T,TD) = 100 * SDD(TD) / SDD(T)
   4. TD(r,T) = b*v/(a-v) mit v(r,T) = log10(DD(r,T)/6.1078)
   5. AF(r,TK) = 10^5 * mw/R* * DD(r,T)/TK; AF(TD,TK) = 10^5 * mw/R* * SDD(TD)/TK 

*)
END_FUNCTION

(* POU Building/HLK/HEAT_INDEX, ST *)
FUNCTION HEAT_INDEX : REAL
VAR_INPUT
	T : REAL;
	RH : REAL;
END_VAR
VAR
	RH2 : REAL;
	T2 : REAL;
END_VAR

(*
version 1.2	2 dec 2007
programmer 	hugo
tested by		tobias

this function calculates the heat index temperature depending on external temperature and Relative humidity

*)
IF RH < 20 OR T < 20 THEN
	Heat_index := T;
ELSE
	RH2 := RH * RH;
	T := C_to_F(T);
	T2 := T * T;
	Heat_index := -42.379 + 2.04901523 * T - 6.83783E-3 * T2
			+ RH * (10.1433127 - 0.22475541 * T + 1.22874E-3 * T2)
			+ RH2 * (8.5282E-4 * T - 5.481717E-2 - 1.99E-6 * T2);
	Heat_index := F_to_C(Heat_index);
END_IF;

(* revision history

hm 27.2.2007		rev 1.1
	deleted unused variables rh3 and T3

hm	2.12.2007		rev 1.2
	changed code for better performance
*)
END_FUNCTION

(* POU Engineering/conversion/C_TO_F, ST *)
FUNCTION C_TO_F : REAL
VAR_INPUT
	celsius : REAL;
END_VAR
VAR
END_VAR

(*
version 1.0	4 aug 2006
programmer 	hugo
tested by		tobias

this function converts celsius  to fahrenheit 

*)
C_to_F := celsius * 1.8 + 32;
END_FUNCTION

(* POU Engineering/conversion/F_TO_C, ST *)
FUNCTION F_TO_C : REAL
VAR_INPUT
	fahrenheit : REAL;
END_VAR
VAR
END_VAR

(*
version 1.1	6. jan 2008
programmer 	hugo
tested BY		tobias

this FUNCTION converts fahrenheit TO celsius

executioin TIME on wago 750-841 = 15us
*)
F_to_C := (fahrenheit -32) * 0.5555555555555;

(* revision history
hm	4. aug 2006		rev 1.0
	original version

hm	6. jan 2008		rev 1.1
	improved performance

*)
END_FUNCTION

(* POU Building/HLK/HEAT_METER, ST *)
FUNCTION_BLOCK HEAT_METER
VAR_INPUT
	TF, TR : REAL;
	LPH : REAL;
	E : BOOL;
	RST : BOOL;
END_VAR
VAR_INPUT CONSTANT
	CP : REAL;
	Density : REAL;
	Content : REAL;
	Pulse_Mode : BOOL;
	Return_meter : BOOL;
	AVG_time : TIME := T#5s;
END_VAR
VAR_OUTPUT
	C : REAL;
END_VAR
VAR_IN_OUT
	Y : REAL;
END_VAR
VAR
	tx, last : DWORD;
	int1 : FT_INT2;
	edge : BOOL;
	x: REAL;
	init: BOOL;
	y_last: REAL;
END_VAR

(*
version 1.6	8. feb. 2009
programmer 	hugo
tested by		oscat

Heat meter measures the heat transfer of water of a mixture of water and another component.
The inputs are foreward temperature and reverse temperature.
the additional component is specified with its parameters density, Specific heat capacity and content in %.
an input e anables the measurement while it can be configured to be based on X liters / pulse or in liters / hour.
the output Y is in Joule.

*)
IF rst THEN
	int1(rst := TRUE);
	int1.rst := FALSE;
	C := Y := 0;
ELSIF e THEN
	X := (WATER_DENSITY(SEL(return_meter, TF, TR), FALSE) * (WATER_ENTHALPY(TF) - WATER_ENTHALPY(TR)) * (1-content) + CP * Density * content*(TF-TR));
	IF pulse_mode THEN
		IF NOT edge THEN Y := Y + X * LPH; END_IF;
	ELSE
		int1(in := X * LPH / 3600.0, out_min := 0, out_max := 3E38);
		Y := int1.Out;
	END_IF;
END_IF;

(* store the value of e *)
edge := e;

(* read system_time *)
tx := T_PLC_MS();

(* only init at startup necessary *)
IF NOT init THEN
	init := TRUE;
	last := tx;
END_IF;

(* calculate the current consumption *)
IF (tx - last >= TIME_TO_DWORD(AVG_TIME)) AND (avg_time > T#0s) THEN
	last := tx;
	C := (Y - Y_last) * 3.6/DWORD_TO_REAL(TIME_TO_DWORD(AVG_TIME));
	Y_last := Y;
END_IF;



(* revision history
hm	16. nov. 2007	rev 1.0
	original version

hm	24. dec. 2007	rev 1.1
	added config variable return_meter
	added output C for current consumption

hm	6. mar. 2008	rev 1.2
	corrected an error in pulse mode

hm	16. mar. 2008	rev 1.3
	added type conversion to avoid warnings under codesys 3.0

hm	21. oct. 2008	rev 1.4
	improved code

hm	6. nov. 2008	rev 1.5
	changed to FT_INT2 to avoid overrun at hig values

hm	8. feb. 2009	rev 1.6
	changes Y to be I/O
*)
END_FUNCTION_BLOCK

(* POU Engineering/control/FT_INT2, ST *)
FUNCTION_BLOCK FT_INT2
VAR_INPUT
	IN : REAL;
	K : REAL := 1;
	RUN : BOOL := 1;
	RST : BOOL;
	OUT_MIN : REAL := -1E37;
	OUT_MAX : REAL := 1E37;
END_VAR
VAR_OUTPUT
	OUT : REAL;
	LIM : BOOL;
END_VAR
VAR
	integ: INTEGRATE;
	ix : REAL;
	val : REAL2;
END_VAR


(*
version 1.1	5. nov. 2008
programmer 	hugo
tested by	oscat

FT_int2 is an integrator with input IN and factor K.
integration is only done while run = true, if run is false integration is stopped and the out remains at the last value.
if run is left unconnected, run is considered true by the function block.
the out_min and out_max values can be set to ,imit the output value range. 
the default for K is 1.
FT_INT2 has double presision accuracy (14 digits).


*)
IF RST THEN
	val := R2_SET(0);
	out := 0;
ELSE
	integ(X := IN, E := RUN, K := K, Y := ix);
	val := R2_ADD(val, ix);
	ix := 0;
	OUT := val.RX;
END_IF;

(* check output for limits *)
IF out > OUT_MIN AND out < OUT_MAX THEN
	LIM := FALSE;
ELSE
	OUT := LIMIT(OUT_MIN, OUT, OUT_MAX);
	val := R2_SET(OUT);
	LIM := TRUE;
END_IF;



(*	revision history
hm	2. jun. 2008	rev 1.0
	original version

hm	5. nov. 2008	rev 1.1
	rewritten code using integrate
*)
END_FUNCTION_BLOCK

(* POU Engineering/control/INTEGRATE, ST *)
FUNCTION_BLOCK INTEGRATE
VAR_INPUT
	E : BOOL := TRUE;
	X : REAL;
	K : REAL := 1;
END_VAR
VAR_IN_OUT
	Y : REAL;
END_VAR
VAR
	X_last : REAL;
	init: BOOL;
	last: DWORD;
	tx: DWORD;
END_VAR


(*
version 1.0	3. nov. 2008
programmer 	hugo
tested by	oscat

integrate is a plain integrator with I/O for out.

 
*)
(*read system time *)
tx := T_PLC_MS();

IF NOT init THEN
	init := TRUE;
	X_last := X;
ELSIF E THEN
	Y := (X + X_LAST) * 0.5E-3 * DWORD_TO_REAL(tx-last) * K + Y;
	X_last := X;
END_IF;
last := tx;



(*
hm 	3. nov. 2008	rev 1.0
original version
	
*)
END_FUNCTION_BLOCK

(* POU Mathematical/Double Precision/R2_SET, ST *)
FUNCTION R2_SET : REAL2
VAR_INPUT
	X : REAL;
END_VAR
VAR
END_VAR

(*
version 1.0	21. mar. 2008
programmer 	hugo
tested by		tobias

R2_set sets a double precision real to a single real value.

*)
R2_SET.RX := X;
R2_SET.R1 := 0;


(* revision history
hm	2. jun. 2008	rev 1.0
	original version

*)
END_FUNCTION

(* POU Building/HLK/WATER_DENSITY, ST *)
FUNCTION WATER_DENSITY : REAL
VAR_INPUT
	T : REAL;
	Sat : BOOL;
END_VAR
VAR CONSTANT
	a0 : REAL := 999.83952;
	a1 : REAL := 16.952577;
	a2 : REAL := -7.9905127E-3;
	a3 : REAL := -4.6241757E-5;
	a4 : REAL := 1.0584601E-7;
	a5 : REAL := -2.8103006E-10;
	b  : REAL := 0.0168872;
END_VAR
VAR
	T2: REAL;
	T4: REAL;
END_VAR


(*
version 1.1	2 dec 2007
programmer 	hugo
tested by		tobias

this function calculates the water density for air free water between 0 and 100 deg C
while sat is false the denisty is calculated for air free water and when sat = true
the calculation is performed for water saturated with air.

*)
T2 := T * T;
T4 := T2 * T2;

(* original code changed for performance
Water_density := (a0 + a1*T + a2*EXPT(T,2) + a3*EXPT(t,3) + a4*EXPT(t,4) + a5*EXPT(t,5)) / (1 + b*T);
*)
Water_density := (a0 + a1*T + a2*T2 + a3*T2*T + a4*T4 + a5*T4*T) / (1 + b*T);

IF sat THEN Water_density := Water_density - 0.004612 + 0.000106 * T; END_IF;


(* revision history

hm	13.9.2007		rev 1.0
	original version

hm	2.12.2007		rev 1.1
	changed code for better performance
*)

(*
    °C - die Celsius-Temperatur in Grad Celsius
    v – das spezifische Volumen in Kubikdezimeter je Kilogramm dm³/kg
    h – die spezifische Enthalpie in Kilojoule je Kilogramm 	kJ/kg
    u – die spezifische Innere Energie in Kilojoule je Kilogramm 	kJ/kg
    s – die spezifische Entropie in Kilojoule je Kilogramm mal Kelvin 	kJ/(kg·K)
    cp - die spezifische Wärmekapazität bei konstantem Druck in Kilojoule je Kilogramm mal Kelvin 	kJ/(kg·K)
    Y – Volumenausdehnungskoeffizient in 10-3 durch Kelvin  10-3/K
    L – Wärmeleitfähigkeit in Milliwatt je Meter mal Kelvin  mW / (m·K) 
    n – Viskosität in Mikropascal mal Sekunde uPa·s 	
    s ? – Oberflächenspannung in Millinewton je Meter  mN/m


°C 		v 				h 			u 		s 			cp 		Y 		L		n		s	
-20		1,006580	
0 		1,000160 		0,06 		-0,04 	-0,0001 	4,228 	-0,080 	561,0 	1792 	75,65
4		1,000028
5 		1,0000 		21,1 		21,0 	0,076 		4,200 	0,011 	570,6 	1518 	74,95
10 		1,0003 		42,1 		42,0 	0,151 		4,188 	0,087 	580,0 	1306 	74,22
15 		1,0009 		63,0 		62,9 	0,224 		4,184 	0,152 	589,4 	1137 	73,49
20 		1,001797 		83,9 		83,8 	0,296 		4,183 	0,209 	598,4 	1001 	72,74
25 		1,0029 		104,8 		104,7 	0,367 		4,183 	0,259 	607,2 	890,4 	71,98
30 		1,0044 		125,8 		125,7 	0,437 		4,183 	0,305 	615,5 	797,7 	71,20
35 		1,0060 		146,7 		146,6 	0,505 		4,183 	0,347 	623,3 	719,6 	70,41
40 		1,007842 		167,58 	167,5 	0,572 		4,182 	0,386 	630,6 	653,3 	69,60
45 		1,0099 		188,5 		188,4 	0,638 		4,182 	0,423 	637,3 	596,3 	68,78
50 		1,0121 		209,4 		209,3 	0,704 		4,181 	0,457 	643,6 	547,1 	67,95
60 		1,017089 		251,2 		251,1 	0,831 		4,183 	0,522 	654,4 	466,6 	66,24
70 		1,0227 		293,1 		293,0 	0,955 		4,187 	0,583 	663,1 	404,1 	64,49
80 		1,029027 		335,0 		334,9 	1,075 		4,194 	0,640 	670,0 	354,5 	62,68
90 		1,0359 		377,0 		376,9 	1,193 		4,204 	0,696 	675,3 	314,6 	60,82
99,63 	1,0431 		417,5 		417,4 	1,303 		4,217 	0,748 	679,0 	283,0 	58,99
100	1,043453		419,1

Stoffdaten von Wasser Quelle Wickipedia

*)
END_FUNCTION

(* POU Building/HLK/WATER_ENTHALPY, ST *)
FUNCTION WATER_ENTHALPY : REAL
VAR_INPUT
	T : REAL;
END_VAR
VAR
	Pts : INT := 11;
	data : ARRAY[1..20, 0..1] OF REAL := 0,0.06, 10,42.1, 20,83.9, 30,125.8, 40,167.58, 50,209.4, 60,251.2, 70,293.1, 80,335.0, 90, 377.0, 100,419.1 ;
END_VAR

(*
version 1.0	29 oct 2007
programmer 	hugo
tested by		tobias

water_enthalpy calculates the enthalpy of liquid water from 0..100 °C 

*)
WATER_ENTHALPY := LINEAR_INT(T, Data, Pts);


(* revision history

hm	29.10.2007	rev 1.0
	original version

*)

(*
    °C - die Celsius-Temperatur in Grad Celsius
    v – das spezifische Volumen in Kubikdezimeter je Kilogramm dm³/kg
    h – die spezifische Enthalpie in Kilojoule je Kilogramm 	kJ/kg
    u – die spezifische Innere Energie in Kilojoule je Kilogramm 	kJ/kg
    s – die spezifische Entropie in Kilojoule je Kilogramm mal Kelvin 	kJ/(kg·K)
    cp - die spezifische Wärmekapazität bei konstantem Druck in Kilojoule je Kilogramm mal Kelvin 	kJ/(kg·K)
    Y – Volumenausdehnungskoeffizient in 10-3 durch Kelvin  10-3/K
    L – Wärmeleitfähigkeit in Milliwatt je Meter mal Kelvin  mW / (m·K) 
    n – Viskosität in Mikropascal mal Sekunde uPa·s 	
    s ? – Oberflächenspannung in Millinewton je Meter  mN/m


°C 		v 				h 			u 		s 			cp 		Y 		L		n		s	
-20		1,006580	
0 		1,000160 		0,06 		-0,04 	-0,0001 	4,228 	-0,080 	561,0 	1792 	75,65
4		1,000028
5 		1,0000 		21,1 		21,0 	0,076 		4,200 	0,011 	570,6 	1518 	74,95
10 		1,0003 		42,1 		42,0 	0,151 		4,188 	0,087 	580,0 	1306 	74,22
15 		1,0009 		63,0 		62,9 	0,224 		4,184 	0,152 	589,4 	1137 	73,49
20 		1,001797 		83,9 		83,8 	0,296 		4,183 	0,209 	598,4 	1001 	72,74
25 		1,0029 		104,8 		104,7 	0,367 		4,183 	0,259 	607,2 	890,4 	71,98
30 		1,0044 		125,8 		125,7 	0,437 		4,183 	0,305 	615,5 	797,7 	71,20
35 		1,0060 		146,7 		146,6 	0,505 		4,183 	0,347 	623,3 	719,6 	70,41
40 		1,007842 		167,58 	167,5 	0,572 		4,182 	0,386 	630,6 	653,3 	69,60
45 		1,0099 		188,5 		188,4 	0,638 		4,182 	0,423 	637,3 	596,3 	68,78
50 		1,0121 		209,4 		209,3 	0,704 		4,181 	0,457 	643,6 	547,1 	67,95
60 		1,017089 		251,2 		251,1 	0,831 		4,183 	0,522 	654,4 	466,6 	66,24
70 		1,0227 		293,1 		293,0 	0,955 		4,187 	0,583 	663,1 	404,1 	64,49
80 		1,029027 		335,0 		334,9 	1,075 		4,194 	0,640 	670,0 	354,5 	62,68
90 		1,0359 		377,0 		376,9 	1,193 		4,204 	0,696 	675,3 	314,6 	60,82
99,63 	1,0431 		417,5 		417,4 	1,303 		4,217 	0,748 	679,0 	283,0 	58,99
100	1,043453		419,1

Stoffdaten von Wasser Quelle Wickipedia

Wasser hat unter Normaldruck seine größte Dichte von 1000 Kilogramm pro Kubikmeter bei 3,98 °C und zeigt damit eine Dichteanomalie. 
Diese besteht darin, dass sich Wasser unterhalb von 3,98 °C bei weiterer Temperaturverringerung, auch beim Wechsel zum festen 
Aggregatzustand, wieder ausdehnt, was man nur von wenigen Stoffen kennt. Die derzeit genauesten publizierten Werte für die maximale 
Dichte liegen bei (999,974950 ± 0,00084) kg/m³ und bei (3,983 ± 0,00067) °C für die Temperatur, bei der dieser Wert erreicht wird. 
Die Werte stellen einen Mittelwert der von verschiedenen physikalischen Instituten veröffentlichten Zahlen dar (Stand 2001).

Die Berechnung der Dichte von luftfreiem Wasser DLF in Abhängigkeit von der Temperatur T ([T] = °C) kann mit Hilfe der folgenden 
Virialgleichung erfolgen:
: \frac{D_{\rm LF}}{\rm g/l} = \frac{a_0 + a_1 T + a_2 T^2 + a_3 T^3 + a_4 T^4 + a_5 T^5}{1 + b T}.
mit den Koeffizienten: a0 = 999,83952; a1 = 16,952577 (°C)-1; a2 = -7,9905127·10-3 (°C)-2; a3 = -4,6241757·10-5 (°C)-3; 
a4 = 1,0584601·10-7 (°C)-4; a5 = -2,8103006·10-10 (°C)-5 und b = 0,0168872. 
Für die Berechnung der Dichte von luftgesättigtem Wasser korrigiert man den Wert nach 
DLG/(g/l) = DLF/(g/l) - 0,004612 + 0,000106 (°C)-1·T. (Quelle: PTB-Mitteilungen 100/3-90)

*)
END_FUNCTION

(* POU Mathematical/functions/LINEAR_INT, ST *)
FUNCTION LINEAR_INT : REAL
VAR_INPUT
	X : REAL;
	XY : ARRAY[1..20,0..1] OF REAL;
	Pts : INT;
END_VAR
VAR
	i : INT;
END_VAR

(*
	version 1.1	27 dec 2007
	programmer 	oscat
	tested BY		oscat

LINEAR_INT calculates an output based on a linear interpolation of up to 20 coordinates given in an array
the input coordinates have to start at the lowest array position and must be sorted ba ascending X values.

*)
(*make sure n is bound within the array size *)
pts := MIN(pts,20);

(* calculate the linear segement interpolation *)
i := 2;
(* search for segment and calculate output
	below and above the defined segments we interpolate the last segment *)
WHILE (i < pts) AND (XY[i,0] < X) DO
	i := i + 1;
END_WHILE;

(* calculate the output value on the corresponding segment coordinates *)
LINEAR_INT := ((XY[i,1] - XY[i-1,1]) * X - XY[i,1] * XY[i-1,0] + XY[i-1,1] * XY[i,0]) / (XY[i,0] - XY[i-1,0]);

(* revision history
hm	7. oct 2007		rev 1.0
	original version

hm	27 dec 2007		rev 1.1
	changed code for better performance
*)
END_FUNCTION

(* POU Building/HLK/HEAT_TEMP, ST *)
FUNCTION_BLOCK HEAT_TEMP
VAR_INPUT
	T_EXT : REAL;
	T_INT : REAL;
	OFFSET : REAL;
	T_REQ : REAL;
END_VAR
VAR_INPUT CONSTANT
	TY_MAX : REAL := 70;
	TY_MIN : REAL := 25;
	TY_CONFIG : REAL := 70;
	T_INT_CONFIG : REAL := 20;
	T_EXT_CONFIG : REAL := -15;
	T_DIFF : REAL := 10;
	C : REAL := 1.33;
	H : REAL := 3;
END_VAR
VAR_OUTPUT
	TY : REAL;
	HEAT : BOOL;
END_VAR
VAR
	tr : REAL;
	tx: REAL;
END_VAR

(*
version 1.1	26. sep. 2008
programmer 	hugo
tested by	oscat

Heat_Temp calculates a heat characteristic based on the formula: tv=ti+(tvmax-ti)*((ti-tau)/(ti-taumin))^(1/n)
while
tv necessary heating temperature.
ti internal room temperature (20°C)
tau current external temperature
taumin external temperature to determine characteristics
C exponent for heating system (normally 1,33 or 1,1 for floor heating)

The two additional inputs TY_min and TY_max set limits for the output TY, while an offset inputs allows to rise or lower the room temperature.

*)
tr := T_INT + OFFSET;
tx := (tr - T_EXT) / (T_INT_CONFIG - T_EXT_CONFIG);

IF T_EXT + H > tr THEN
	TY := 0;
ELSE
	TY := LIMIT(TY_MIN, tr + T_DIFF / 2 * tx + (TY_CONFIG - T_DIFF/2 - tr) * EXPT(tx, 1 / C), TY_MAX);
END_IF;

TY := MAX(TY, T_REQ);
HEAT := TY > 0;


(*

tv=ti+(tvmax-ti)*((ti-tau)/(ti-taumin))^(1/n)

tv aktuelle Vorlauftemp.
ti Raumtemperatur innen (20°C)
tau aktuelle Außentemperatur
taumin minimale Außentemperatur -12°C oder -15°C
n Heizkörperexponent (meistens 1,33)
Fußbodenheizung = 1,1
Wandheizung 1,3

Normen z. B. DIN 4703, DIN 4725 oder die Literatur, z. B Recknagel Abschnitt 1.3.5.

*)


(* revision history
hm	27. jan. 2008	rev 1.0
	original version

hm	26. sep. 2008	rev 1.1
	moved T_INT from config to Input
	added config variable H
	corrected error in formula
*)
END_FUNCTION_BLOCK

(* POU Building/HLK/LEGIONELLA, ST *)
FUNCTION_BLOCK LEGIONELLA
VAR_INPUT
	manual : BOOL;
	temp_boiler : REAL;
	temp_return : REAL := 100;
	DT_in: DT;
	rst : BOOL;
END_VAR
VAR_INPUT CONSTANT
	T_start: TOD := tod#03:00:00;
	day : INT := 7;
	temp_set : REAL := 70;
	temp_offset : REAL := 10;
	temp_hys : REAL := 5;
	t_max_heat: TIME := t#10m;
	t_max_ret : TIME := t#10m;
	tp_0: TIME := t#5m;
	tp_1: TIME := t#5m;
	tp_2: TIME := t#5m;
	tp_3: TIME := t#5m;
	tp_4: TIME := t#5m;
	tp_5: TIME := t#5m;
	tp_6: TIME := t#5m;
	tp_7: TIME := t#5m;
END_VAR
VAR_OUTPUT
	Heat : BOOL;
	pump : BOOL;
	valve0 : BOOL;
	valve1 : BOOL;
	valve2 : BOOL;
	valve3 : BOOL;
	valve4 : BOOL;
	valve5 : BOOL;
	valve6 : BOOL;
	valve7 : BOOL;
	run: BOOL;
	Status : BYTE;
END_VAR
VAR
	X1: timer_1;
	x2: sequence_8;
	x3: hyst_1;
	init: BOOL;
END_VAR

(*
version 1.2	23. oct 2008
programmer 	oscat
tested by	oscat

Legionella is a complete sequencer for up to 8 hot water lines that need to be sterilzed periodically.
legionella needs a DT input with the appropriate time, usually gererated by the rtc of the system. for system independence this time is connected externally.
T_start is the time when sterilazation should be started and day is the day_of_week when it should be performed (1=Monday and 7=sunday).
so sterilazation is autioimatically performed once a week at a specified time.
temp_set and temp_hys and temp_offset specify the boiler temperatur nedded for sterilization. as a defaut Temp_set is set to 70 deg C and Temp_hys is set to 5 deg C and temp_offset is 10 deg C.
a temp boiler input reads the boiler temperature of the hot water tank.
after a start pulse is gererated by the weekly timer or a manual test input the sequence is started:
1. the boiler is heated to temp_set + temp_offset + temp_hys = 85 deg C unless chaged at setup.
	the heat output is turned on and tells the heater to turn heating on. if the temp is not reached for a time of t_max_heat (10 min) the error output is set and the sequence is stopped.
2. after the specified temperature is reached, the output valve0 and pump is turned on and starts sterilization of line0 until temp_return has reached temp_set and continues to sterilize for a time of tp_0 (5 min default).
	if tmep_set is not reached at the temp_return_input then the error output is set and the sequence will be stopped.
	if there is no temp sensor for temp_return (the temperature at the return point for the circulation pump pls set this imput to a value greater then temp_set (by default use 100 deg C).
	in this case sterilization is performed for the default times without monitoring the return temp.
3. this sequence is repeated for up to valves.

connection scheme:

temp_boiler:	input oif the boiler temperature sensor.
temp_hys:		config value for the heater hysteresis, preset to 5 deg C.
temp_offset:	config value for the heater temp_offset against temp_set, preset to 10 deg C.
temp_set:		config value for the specified sterilization temperature, preset to 70 deg C.
temp_return:	input of the circulation return line temperature sensor, if not availabe set this value to 100 deg C.
manual:		manual input to start the sterilization by hand for diagnostic purposes, rising edge active, leave low for automatic operation.
DT_in:			date,time input supplied by a external real time clock.
T_start:		time of day when the sterilization should be started.
day:			config value for day of week when the process should be started, preset to sunday.
t_max_hest:	tmax time to be needed for the heater to heat the hot water tank to the specified value, preset to 10 min.

*)
(* startup initialization *)
IF NOT init THEN
	init := TRUE;
	X1.day := SHR(BYTE#128,day);
	X1.start := T_start;
	X3.low := Temp_offset + temp_set;
	X3.high := Temp_hys + X3.low;
	X2.wait0 := T_max_heat;
	X2.delay0 := TP_0;
	X2.delay1 := TP_1;
	X2.delay2 := TP_2;
	X2.delay3 := TP_3;
	X2.delay4 := TP_4;
	X2.delay5 := TP_5;
	X2.delay6 := TP_6;
	X2.delay7 := TP_7;
	X2.wait1 := T_max_ret;
	X2.wait2 := T_max_ret;
	X2.wait3 := T_max_ret;
	X2.wait4 := T_max_ret;
	X2.wait5 := T_max_ret;
	X2.wait6 := T_max_ret;
	X2.wait7 := T_max_ret;
	X2();
END_IF;

(* oerational code *)
X1(DTi := DT_in);
IF X1.Q OR manual OR x2.run THEN
	X3(in := temp_boiler);
	X2.in0 := X3.Q OR x3.win;
	X2.in1 := temp_return >= temp_set;
	X2.in2 := x2.in1;
	X2.in3 := x2.in1;
	X2.in4 := x2.in1;
	X2.in5 := x2.in1;
	X2.in6 := x2.in1;
	X2.in7 := x2.in1;
	X2.rst := rst;
	X2(start := X1.Q OR manual);
	run := x2.run;
	pump := x2.any;
	Heat := NOT X3.Q AND x2.run;
	valve0 := X2.Q0;
	valve1 := X2.Q1;
	valve2 := X2.Q2;
	valve3 := X2.Q3;
	valve4 := X2.Q4;
	valve5 := X2.Q5;
	valve6 := X2.Q6;
	valve7 := X2.Q7;
	pump := X2.any;
	status := X2.status;
ELSE;
	X2(start :=0);
	status := x2.status;
END_IF;

(* revision history

hm 17.jan 2007	rev 1.1
	rewritten to st for higher performance
	changes eeror output to esr compatible status output

hm	23. 10.2008	rev 1.2
	update code to use new version of timer_1
*)
END_FUNCTION_BLOCK

(* POU Logic/generators/SEQUENCE_8, ST *)
FUNCTION_BLOCK SEQUENCE_8
VAR_INPUT
	in0 : BOOL := TRUE;
	in1 : BOOL := TRUE;
	in2 : BOOL := TRUE;
	in3 : BOOL := TRUE;
	in4 : BOOL := TRUE;
	in5 : BOOL := TRUE;
	in6 : BOOL := TRUE;
	in7 : BOOL := TRUE;
	start : BOOL;
	rst : BOOL;
	wait0 : TIME;
	delay0 : TIME;
	wait1 : TIME;
	delay1 : TIME;
	wait2 : TIME;
	delay2 : TIME;
	wait3 : TIME;
	delay3 : TIME;
	wait4 : TIME;
	delay4 : TIME;
	wait5 : TIME;
	delay5 : TIME;
	wait6 : TIME;
	delay6 : TIME;
	wait7 : TIME;
	delay7 : TIME;
END_VAR
VAR_INPUT CONSTANT
	stop_on_error : BOOL;
END_VAR
VAR_OUTPUT
	Q0 : BOOL;
	Q1 : BOOL;
	Q2 : BOOL;
	Q3 : BOOL;
	Q4 : BOOL;
	Q5 : BOOL;
	Q6 : BOOL;
	Q7 : BOOL;
	any : BOOL;
	run: BOOL;
	step : INT := -1;
	status : BYTE;
END_VAR
VAR
	last : TIME;
	edge : BOOL;
	tx: TIME;
	init: BOOL;
END_VAR

(*
version 1.4	17 sep 2007
programmer 	oscat
tested by		hans

sequence_8 enables run when a low to high transition is present on start.
a low to high transition on start will restart the sequencer at any time while a rst will hold the sequencer in reset while true.
after run is enabled with a rising edge on start the sequencer waits for wait0 on in0 to enable q0 which stays on for delay0.
the next cycle starts with wait1, continues with delay 1 and so on...
if an edge is not detected during the wait period, the sequencer will then display the error number on the status output.
The status numbers are 1 .. 8 for erros in step 0..7.
after the last step that sets q7, the sequencer leaves q7 on for delay7 and then resets to the initial state.
a step output will indicate the current step of the sequencer and will also be present with a fault condition.
after the first output is turened on the sequencer switches from q0 to q1 and so on, at any time there is only one output enabled.
if an input signal is not detected during a wait period, the sequencer will display the error number ( 1 for in0, 2 for in1 .... ).
when an error is present and the config variable stop_on_error is set then the sequencer will stop. otherwise it will continue.
The status output will also display 110 for waiting and 111 sequece running.

*)
(* read sps timer *)
tx := DWORD_TO_TIME(T_PLC_MS());

(* initialize on startup *)
IF NOT init THEN
	last := tx;
	init := TRUE;
	status := 110;
END_IF;

(* asynchronous reset *)
IF rst THEN
	step := -1;
	Q0 := 0;
	Q1 := 0;
	Q2 := 0;
	Q3 := 0;
	Q4 := 0;
	Q5 := 0;
	Q6 := 0;
	Q7 := 0;
	status := 110;
	run := 0;

(* edge on start input restarts the sequencer *)
ELSIF start AND NOT edge THEN
	step := 0;
	last := tx;
	status := 111;
	Q0 := 0;
	Q1 := 0;
	Q2 := 0;
	Q3 := 0;
	Q4 := 0;
	Q5 := 0;
	Q6 := 0;
	Q7 := 0;
	run := 1;
END_IF;
edge := start;

(* check if stop on error is necessary *)
IF status > 0 AND status < 100 AND stop_on_error THEN RETURN; END_IF;

(* sequence is running *)
IF run AND step = 0 THEN
	IF NOT q0 AND in0 AND tx - last <= wait0 THEN
		Q0 := TRUE;
		last := tx;
	ELSIF NOT q0 AND tx - last > wait0 THEN
		status := 1;
		run := FALSE;
	ELSIF q0 AND tx - last >= delay0 THEN
		step := 1;
		last := tx;
	END_IF;
END_IF;
IF run AND step = 1 THEN
	IF NOT q1 AND in1 AND tx - last <= wait1 THEN
		Q0 := FALSE;
		Q1 := TRUE;
		last := tx;
	ELSIF NOT q1 AND Tx - last > wait1 THEN
		status := 2;
		q0 := FALSE;
		run := FALSE;
	ELSIF q1 AND tx - last >= delay1 THEN
		step := 2;
		last := tx;
	END_IF;
END_IF;
IF run AND step = 2 THEN
	IF NOT q2 AND in2 AND tx - last <= wait2 THEN
		Q1 := FALSE;
		Q2 := TRUE;
		last := tx;
	ELSIF NOT q2 AND Tx - last > wait2 THEN
		status := 3;
		q1 := FALSE;
		run := FALSE;
	ELSIF q2 AND tx - last >= delay2 THEN
		step := 3;
		last := tx;
	END_IF;
END_IF;
IF run AND step = 3 THEN
	IF NOT q3 AND in3 AND tx - last <= wait3 THEN
		Q2 := FALSE;
		Q3 := TRUE;
		last := tx;
	ELSIF NOT q3 AND Tx - last > wait3 THEN
		status := 4;
		q2 := FALSE;
		run := FALSE;
	ELSIF q3 AND tx - last >= delay3 THEN
		step := 4;
		last := tx;
	END_IF;
END_IF;
IF run AND step = 4 THEN
	IF NOT q4 AND in4 AND tx - last <= wait4 THEN
		Q3 := FALSE;
		Q4 := TRUE;
		last := tx;
	ELSIF NOT q4 AND Tx - last > wait4 THEN
		status := 5;
		q3 := FALSE;
		run := FALSE;
	ELSIF q4 AND tx - last >= delay4 THEN
		step := 5;
		last := tx;
	END_IF;
END_IF;
IF run AND step = 5 THEN
	IF NOT q5 AND in5 AND tx - last <= wait5 THEN
		Q4 := FALSE;
		Q5 := TRUE;
		last := tx;
	ELSIF NOT q5 AND Tx - last > wait5 THEN
		status := 6;
		q4 := FALSE;
		run := FALSE;
	ELSIF q5 AND tx - last >= delay5 THEN
		step := 6;
		last := tx;
	END_IF;
END_IF;
IF run AND step = 6 THEN
	IF NOT q6 AND in6 AND tx - last <= wait6 THEN
		Q5 := FALSE;
		Q6 := TRUE;
		last := tx;
	ELSIF NOT q6 AND Tx - last > wait6 THEN
		status := 7;
		q5 := FALSE;
		run := FALSE;
	ELSIF q6 AND tx - last >= delay6 THEN
		step := 7;
		last := tx;
	END_IF;
END_IF;
IF run AND step = 7 THEN
	IF NOT q7 AND in7 AND tx - last <= wait7 THEN
		Q6 := FALSE;
		Q7 := TRUE;
		last := tx;
	ELSIF NOT q7 AND Tx - last > wait7 THEN
		status := 8;
		q6 := FALSE;
		run := FALSE;
	ELSIF q7 AND tx - last >= delay7 THEN
		step := -1;
		Q7 := FALSE;
		Run := FALSE;
		status := 110;
	END_IF;
END_IF;
any := q0 OR q1 OR q2 OR q3 OR q4 OR q5 OR q6 OR q7;

(*
hm 1.10.06		rev 1.1
	corrected delay logic to be after event and not before
	added any output

hm 1.12.06		rev 1.2
	corrected failure in sequence logic.
	added init at startup to prevent from initial statuss after start.

hm 17.1.2007		rev 1.3
	changed output fault to status for better compatibility with other modules (ESR)
	added stop on error functionality and setup variable
	default for inputs in0..7 is true.
	renames variable state to step

hm	17.sep 2007		rev 1.4
	replaced time() with T_PLC_MS() for compatibility reasons

*)
END_FUNCTION_BLOCK

(* POU Engineering/control/HYST_1, ST *)
FUNCTION_BLOCK HYST_1
VAR_INPUT
	In : REAL;
	high : REAL;
	low : REAL;
END_VAR
VAR_OUTPUT
	Q : BOOL;
	win : BOOL;
END_VAR
VAR
END_VAR

(*
version 1.1	2. jun. 2008
programmer 	hugo
tested BY	oscat

this hysteresis function switches the output high if the input signal reaches obove high and will switch to low when the input falls back below low value.
a separate output mid is set if the input stays between low and high value.

*)
IF in < low THEN
	Q := FALSE;
	win := FALSE;
ELSIF in > high THEN
	Q := TRUE;
	win := FALSE;
ELSE
	win := TRUE;
END_IF;

(* code used for rev 1.0
IF Q THEN
	IF in < low THEN q := FALSE; END_IF;
ELSE
	IF in > high THEN q := TRUE; END_IF;
END_IF;
win := in > low AND in < high;
*)


(* revision history
hm		4.  aug. 2006	rev 1.0
	original version

hm		2. jun. 2008	rev 1.1
	improved performance
*)
END_FUNCTION_BLOCK

(* POU Building/HLK/T_AVG24, ST *)
FUNCTION_BLOCK T_AVG24
VAR_INPUT
	TS : INT;
	DTI : DT;
	RST : BOOL;
END_VAR
VAR_INPUT CONSTANT
	T_FILTER : TIME := T#10m;
	SCALE : REAL := 1.0;
	OFS : REAL;
END_VAR
VAR_OUTPUT
	TA : REAL;
	TP : BOOL;
END_VAR
VAR_IN_OUT
	T24 : REAL;
	T24_MAX : REAL;
	T24_MIN : REAL;
END_VAR
VAR
	samples : ARRAY[0..47] OF INT;
	pos : INT;
	init: BOOL;
	ft1 : FILTER_I;
	sum : DINT;
	last: DT;
END_VAR
VAR_TEMP
	tmp_max : INT;
	tmp_min : INT;
	i: INT;
END_VAR

(*
version 1.0	8. feb. 2009
programmer 	hugo
tested by	oscat

this function calculates the averaged daytime temperature by taking 48 samples over one day.
a trigger tp will be true for one cycle when the output is updated.
using the input scale the outputs can be adjusted to different scales.

*)
(* first filter the sensor readings *)
ft1(X := TS, T := T_FILTER);

IF rst OR NOT init THEN
	init := TRUE;
	IF T24 = -1000 THEN t24 := INT_TO_REAL(ft1.Y) / 10.0; END_IF;
	FOR pos := 0 TO 47 DO
		samples[pos] := REAL_TO_INT(T24 * 10.0);
	END_FOR;
	pos := 0;
	sum := INT_TO_DINT(samples[0]) * 48;
	(* calculate the output value *)
	TA := (INT_TO_REAL(ft1.Y)/10.0 + OFS) * SCALE;
	T24 := (DINT_TO_REAL(sum) / 480.0 + OFS) * SCALE;
	tp := TRUE;
ELSIF DT_TO_DWORD(dti) / 60 MOD 30 = 0 AND DTI > last THEN
	(* make sure we onlyexecute once every 30 mins *)
	last := DTI + T#1m;
	(* sample the temperature every 30 mins and store in ring buffer samples *)
	(* sum always holds the sum of the array *)
	(* subtract the oldest sample from sum *)
	sum := sum - INT_TO_DINT(samples[pos]);
	(* strore the new sample *)
	samples[pos] := ft1.Y;
	(* add the new sample to sum *)
	sum := sum + INT_TO_DINT(samples[pos]);
	(* increment the counter for the next sample *)
	pos := INC1(pos, 48);
	(* calculate the output value *)
	TA := (INT_TO_REAL(ft1.Y)/10.0 + OFS) * SCALE;
	T24 := (DINT_TO_REAL(sum) / 480.0 + OFS) * SCALE;
	(* calculate the min and max over the last 24 hours *)
	tmp_max := -32000;
	tmp_min := 32000;
	FOR i := 0 TO 47 DO
		tmp_max := MAX(tmp_max, samples[i]);
		tmp_min := MIN(tmp_min, samples[i]);
	END_FOR;
	T24_MAX := (INT_TO_REAL(tmp_max) / 10.0 + OFS) * SCALE;
	T24_MIN := (INT_TO_REAL(tmp_min) / 10.0 + OFS) * SCALE;
	tp := TRUE;
ELSE
	tp := FALSE;
END_IF;





(* revision history
hm	3. nov. 2008	rev 1.0
	original version

hm	8. feb. 2009	rev 1.1
	changes sign of OFS
	added outputs t24_min and t24_max

*)
END_FUNCTION_BLOCK

(* POU Engineering/signal processing/SCALE, ST *)
FUNCTION SCALE : REAL
VAR_INPUT
	X : REAL;
	K : REAL;
	O : REAL;
	MX : REAL;
	MN : REAL;
END_VAR
VAR
END_VAR

(*
version 1.0	16. may. 2008
programmer 	hugo
tested by		tobias

Scale is used to translate an input x to output by the formula Y = X*K + O.
at the same time the output is limited to MN and MX.

*)
SCALE := LIMIT(MN, X * K + O, MX);


(* revision history
hm	16. may. 2008		rev 1.0
	original version
*)
END_FUNCTION

(* POU Engineering/signal processing/FILTER_I, ST *)
FUNCTION_BLOCK FILTER_I
VAR_INPUT
	X : INT;
	T : TIME;
END_VAR
VAR_OUTPUT
	Y : INT;
END_VAR
VAR
	Yi : DINT;
	last : DWORD;
	tx: DWORD;
	init: BOOL;
END_VAR

(*
version 1.0	8. nov. 2008
programmer 	hugo
tested by	oscat

FILTER_I is a low pass filter with a programmable time T used for INT format.
 
*)
(* read system time *)
tx := T_PLC_MS();

(* startup initialisation *)
IF NOT init OR T = t#0s THEN
	init := TRUE;
	Yi := INT_TO_DINT(X) * 1000;
ELSE
	(* to increase accuracy of the filter we calculate internal Yi wich is Y * 1000 *)
	Yi := Yi + INT_TO_DINT(X - Y) * DWORD_TO_DINT(tx - last) * 1000 / TIME_TO_DINT(T);
END_IF;
last := tx;
Y := DINT_TO_INT(yi / 1000);



(*
hm 8. nov. 2008	rev 1.0
	original version

*)
END_FUNCTION_BLOCK

(* POU Mathematical/INC1, ST *)
FUNCTION INC1 : INT
VAR_INPUT
	X : INT;
	N : INT;
END_VAR
VAR
END_VAR


(*
version 1.2	23. feb. 2009
programmer 	hugo
tested by	oscat

This is a increment function which increments the variable X by 1 and if N is reached, it begins with 0 instead of N again.
inc1(X,3) will generate 0,1,2,0,1,.....

*)
IF X >= N - 1 THEN
	INC1 := 0;
ELSE
	INC1 := X + 1;
END_IF;


(* this elegant version is 50% slower
INC1 := X := (x + 1) MOD N;
*)



(* revision history
hm	13. oct. 2008	rev 1.0
	original version

hm	22. oct. 2008	rev 1.1
	added statement to return value for compatibility reasons

hm	23. feb. 2009	rev 1.2
 	when inc1 is called with X >= N inc will continue with 0
*)
END_FUNCTION

(* POU Building/HLK/TEMP_EXT, ST *)
FUNCTION_BLOCK TEMP_EXT
VAR_INPUT
	t_ext1 : REAL;
	t_ext2 : REAL;
	t_ext3 : REAL;
	t_ext_config : BYTE := 0;
	dt_in : DT;
END_VAR
VAR_INPUT CONSTANT
	t_ext_min : REAL := -40;
	t_ext_max : REAL := 60;
	t_ext_default : REAL := -10;
	heat_period_start : DATE := D#1970-9-1;
	heat_period_stop : DATE := D#1970-4-30;
	cool_period_start : DATE := D#1970-4-1;
	cool_period_stop : DATE := D#1970-9-30;
	heat_start_temp_day : REAL := 15;
	heat_start_temp_night : REAL := 10;
	heat_stop_temp : REAL := 18;
	cool_start_temp_day : REAL := 26;
	cool_start_temp_night : REAL := 26;
	cool_stop_temp : REAL := 24;
	start_day : TOD := tod#09:00;
	start_night : TOD := tod#21:00;
	cycle_time : TIME := t#10m;
END_VAR
VAR_OUTPUT
	t_ext : REAL;
	heat : BOOL;
	cool : BOOL;
END_VAR
VAR
	tx: TIME;
	last_run: TIME;
	init: BOOL;
	cool_start: DATE;
	cool_stop: DATE;
	heat_start: DATE;
	heat_stop: DATE;
	xdate: DATE;
	day: BOOL;
END_VAR


(*
version 1.2	7. oct. 2008
programmer 	hugo
tested by	oscat

temp_ext measures and processes ext temperature and decides if heating or cooling is needed.

 the measurement of t_ext has 3 inputs which can be configured in different ways:
	t_ext_config = 0 means the ext temp is the avg of the 3 external temperatures, this mode is the default mode.
	t_ext_config = 1 means t_ext1 is used.
	t_ext_config = 2 means t_ext1 is used.
	t_ext_config = 3 means t_ext1 is used.
	t_ext_config = 4 means t_ext_default is used.
	t_ext_config = 5 means the lowest of the 3 external temperatures is used.
	t_ext_config = 6 means the higest externnal temperature is used.
	t_ext_config = 7 means the midlle external temperature is used, if there are only two working, the lowest is used.
	in any config mode, an external temperature higher then t_ext_max or lower then t_ext_min is ignored to prevent from temperatures caused by broken sensors or wires.
	if no external temperature is available, a default value (t_ext_default) is used.
	if you have only one external sensor, connect the 3 inputs to the same sensor, or select the right input with t_ext_config.

heating or cooling is enabled during heating / cooling period when the day or night start temperature is reached for at least the specified delay time and will be disabled after the stop temperature is reached. 
t_ext output can be used by other modules to determine the correct system temperature for heating or cooling.

*)
IF NOT init THEN
	init := TRUE;
	heat_start := SET_DATE(1972,MONTH_OF_DATE(heat_period_start),DAY_OF_MONTH(heat_period_start));
	heat_stop := SET_DATE(1972,MONTH_OF_DATE(heat_period_stop),DAY_OF_MONTH(heat_period_stop));
	cool_start := SET_DATE(1972,MONTH_OF_DATE(cool_period_start),DAY_OF_MONTH(cool_period_start));
	cool_stop := SET_DATE(1972,MONTH_OF_DATE(cool_period_stop),DAY_OF_MONTH(cool_period_stop));
END_IF;

(* read system time *)
tx := DWORD_TO_TIME(T_PLC_MS());

(* for efficiency exit isf this program has been executed less then 1min ago *)
IF tx - last_run < cycle_time THEN RETURN; END_IF;

(* calculate frequently used variables *)
xdate := SET_DATE(1972,MONTH_OF_DATE(DT_TO_DATE(dt_in)),DAY_OF_MONTH(DT_TO_DATE(dt_in)));
day := DT_TO_TOD(dt_in) >= start_day AND  DT_TO_TOD(dt_in) < start_night;

(* read the correct external temperature depending on the t_ext_config setting *)
t_ext := multi_in(t_ext1, t_ext2, t_ext3, t_ext_default, t_ext_min, t_ext_max, t_ext_config);

(* dtermine heating *)
IF (heat_start <= heat_stop AND xdate >= heat_start AND xdate <= heat_stop) OR (heat_start > heat_stop AND (xdate >= heat_start OR xdate <= heat_stop)) THEN
	(* heating period id true check for temperature *)
	IF day AND t_ext <= heat_start_temp_day THEN
		heat := TRUE;
	ELSIF NOT day AND t_ext <= heat_start_temp_night THEN
		heat := TRUE;
	ELSIF t_ext >= heat_stop_temp THEN
		heat := FALSE;
	END_IF;
ELSE
	heat := FALSE;
END_IF;

(* dtermine cooling *)
IF (cool_start <= cool_stop AND xdate >= cool_start AND xdate <= cool_stop) OR (cool_start > cool_stop AND (xdate >= cool_start OR xdate <= cool_stop)) THEN
	(* cooling period is true check for temperature *)
	IF day AND t_ext >= cool_start_temp_day THEN
		cool := TRUE;
	ELSIF NOT day AND t_ext >= cool_start_temp_night THEN
		cool := TRUE;
	ELSIF t_ext <= cool_stop_temp THEN
		cool := FALSE;
	END_IF;
ELSE
	cool := FALSE;
END_IF;

last_run := tx;

(* revision history
hm	6 dec 2006		rev 1.0
	original version

hm	15.9.2007		rev 1.1
	replaced Time() with T_PLC_MS for compatibility and performance reasons

hm	7. oct. 2008	rev 1.2
	changed name of function month to month_of_date

*)
END_FUNCTION_BLOCK

(* POU Engineering/sensor/MULTI_IN, ST *)
FUNCTION MULTI_IN : REAL
VAR_INPUT
	in_1 : REAL;
	in_2 : REAL;
	in_3 : REAL;
	default : REAL;
	in_min : REAL;
	in_max : REAL;
	mode : BYTE;
END_VAR
VAR
	count: INT;
	F1: BOOL;
	F2: BOOL;
	F3: BOOL;
END_VAR

(*

version 1.2	14. oct. 2008
programmer 	oscat
tested by	oscat

multi_in is a signal conditioning function which can be configured in 8 different ways.
it is used to read multiple sensors for the same value and protect the user from broken sensors or invalid data from sensors.

multi_in can be configured in different ways:
	mode = 0 means the the avg of the 3 inputs is used, this mode is the default mode.
	mode = 1 means in_1 is used.
	mode = 2 means in_2 is used.
	mode = 3 means in_3 is used.
	mode = 4 means default is used.
	mode = 5 means the lowest of the 3 external temperatures is used.
	mode = 6 means the higest externnal temperature is used.
	mode = 7 means the midlle input is used, if there are only two working, the lowest input is used.
	mode > 7 ,eans output is 0 at all times.
	in any config mode, an input higher then in_max or lower then in_min is ignored to prevent values from broken sensors or wires.
	if all inputs are higher then in_max or lower then in_min, a default value (default) is used.
*)
F1 :=  in_1 > in_min AND in_1 < in_max;
F2 :=  in_2 > in_min AND in_2 < in_max;
F3 :=  in_3 > in_min AND in_3 < in_max;

CASE mode OF
0:	count := 0;
	IF F1 THEN
		count := count + 1;
		MULTI_IN := in_1;
	ELSE
		MULTI_IN := 0;
	END_IF;
	IF F2 THEN
		count := count + 1;
		MULTI_IN := MULTI_IN + in_2;
	END_IF;
	IF F3 THEN
		count := count + 1;
		MULTI_IN := MULTI_IN + in_3;
	END_IF;
	IF count = 0 THEN
		MULTI_IN := default;
	ELSE
		MULTI_IN := MULTI_IN / count;
	END_IF;

1:	IF F1 THEN MULTI_IN := in_1; ELSE MULTI_IN := default; END_IF;

2:	IF F2 THEN MULTI_IN := in_2; ELSE MULTI_IN := default; END_IF;

3:	IF F3 THEN MULTI_IN := in_3; ELSE MULTI_IN := default; END_IF;

4:	MULTI_IN := default;

5:	IF F1 THEN MULTI_IN := in_1; ELSE MULTI_IN := in_max; END_IF;
	IF F2 AND in_2 < MULTI_IN THEN MULTI_IN := in_2; END_IF;
	IF F3 AND in_3 < MULTI_IN THEN MULTI_IN := in_3; END_IF;
	IF MULTI_IN = in_max THEN MULTI_IN := default; END_IF;

6:	IF F1 THEN MULTI_IN := in_1; ELSE MULTI_IN := in_min; END_IF;
	IF F2 AND in_2 > MULTI_IN THEN MULTI_IN := in_2; END_IF;
	IF F3 AND in_3 > MULTI_IN THEN MULTI_IN := in_3; END_IF;
	IF MULTI_IN = in_min THEN MULTI_IN := default; END_IF;

7:	IF F1 AND F2 AND F3 THEN MULTI_IN := MID3(in_1, in_2, in_3);
	ELSIF F1 AND F2 THEN MULTI_IN := MIN(in_1, in_2);
	ELSIF F1 AND F3 THEN MULTI_IN := MIN(in_1, in_3);
	ELSIF F2 AND F3 THEN MULTI_IN := MIN(in_2, in_3);
	ELSIF F1 THEN MULTI_IN := in_1;
	ELSIF F2 THEN MULTI_IN := in_2;
	ELSIF F3 THEN MULTI_IN := in_3;
	ELSE MULTI_IN := default;
	END_IF;

END_CASE;

(*
hm 1.1.2007			rev 1.1
	changed midr to mid3 function

hm	14. 10. 2008	rev 1.2
	corrected an error for in_3 overrange detection
	improved performance


*)
END_FUNCTION

(* POU Mathematical/MID3, ST *)
FUNCTION MID3 : REAL
VAR_INPUT
	in1 : REAL;
	in2 : REAL;
	in3 : REAL;
END_VAR
VAR
END_VAR

(*
version 1.1	1 jan 2007
programmer 	hugo
tested by		tobias

returns the mid value of 3 real inputs.

*)
IF (in1 <= in2) AND (in1 >= in3) OR (in1 >= in2) AND (in1 <= in3) THEN
	mid3 := in1;
ELSIF (in2 <= in1) AND (in2 >= in3) OR (in2 >= in1) AND (in2 <= in3) THEN
	mid3 := in2;
ELSE
	mid3 := in3;
END_IF;

(*
hm	1.1.2007	rev 1.1
	rewrote the function for better performance

*)
END_FUNCTION

(* POU Building/HLK/WATER_CP, ST *)
FUNCTION WATER_CP : REAL
VAR_INPUT
	T : REAL;
END_VAR
VAR
	Pts : INT := 10;
	data : ARRAY[1..20, 0..1] OF REAL := 0,4.228, 5,4.20, 10,4.188, 15,4.184, 50,4.181, 60,4.183, 70,4.187, 80,4.194, 90,4.204, 100,4.22;
END_VAR

(*
version 1.1	27 dec 2007 
programmer 	hugo
tested by	tobias

water_cp calculates the specific heat capacity of liquid water from 0..100 °C 

*)
WATER_CP := LINEAR_INT(T, Data, Pts);


(* revision history

hm	29.10.2007		rev 1.0
	original version

hm	27. dec 2007	rev 1.1
	increased accuracy

*)

(*
    °C - die Celsius-Temperatur in Grad Celsius
    v – das spezifische Volumen in Kubikdezimeter je Kilogramm dm³/kg
    h – die spezifische Enthalpie in Kilojoule je Kilogramm 	kJ/kg
    u – die spezifische Innere Energie in Kilojoule je Kilogramm 	kJ/kg
    s – die spezifische Entropie in Kilojoule je Kilogramm mal Kelvin 	kJ/(kg·K)
    cp - die spezifische Wärmekapazität bei konstantem Druck in Kilojoule je Kilogramm mal Kelvin 	kJ/(kg·K)
    Y – Volumenausdehnungskoeffizient in 10-3 durch Kelvin  10-3/K
    L – Wärmeleitfähigkeit in Milliwatt je Meter mal Kelvin  mW / (m·K) 
    n – Viskosität in Mikropascal mal Sekunde uPa·s 	
    s ? – Oberflächenspannung in Millinewton je Meter  mN/m


°C 		v 				h 			u 		s 			cp 		Y 		L		n		s	
-20		1,006580	
0 		1,000160 		0,06 		-0,04 	-0,0001 	4,228 	-0,080 	561,0 	1792 	75,65
4		1,000028
5 		1,0000 		21,1 		21,0 	0,076 		4,200 	0,011 	570,6 	1518 	74,95
10 		1,0003 		42,1 		42,0 	0,151 		4,188 	0,087 	580,0 	1306 	74,22
15 		1,0009 		63,0 		62,9 	0,224 		4,184 	0,152 	589,4 	1137 	73,49
20 		1,001797 		83,9 		83,8 	0,296 		4,183 	0,209 	598,4 	1001 	72,74
25 		1,0029 		104,8 		104,7 	0,367 		4,183 	0,259 	607,2 	890,4 	71,98
30 		1,0044 		125,8 		125,7 	0,437 		4,183 	0,305 	615,5 	797,7 	71,20
35 		1,0060 		146,7 		146,6 	0,505 		4,183 	0,347 	623,3 	719,6 	70,41
40 		1,007842 		167,58 	167,5 	0,572 		4,182 	0,386 	630,6 	653,3 	69,60
45 		1,0099 		188,5 		188,4 	0,638 		4,182 	0,423 	637,3 	596,3 	68,78
50 		1,0121 		209,4 		209,3 	0,704 		4,181 	0,457 	643,6 	547,1 	67,95
60 		1,017089 		251,2 		251,1 	0,831 		4,183 	0,522 	654,4 	466,6 	66,24
70 		1,0227 		293,1 		293,0 	0,955 		4,187 	0,583 	663,1 	404,1 	64,49
80 		1,029027 		335,0 		334,9 	1,075 		4,194 	0,640 	670,0 	354,5 	62,68
90 		1,0359 		377,0 		376,9 	1,193 		4,204 	0,696 	675,3 	314,6 	60,82
99,63 	1,0431 		417,5 		417,4 	1,303 		4,217 	0,748 	679,0 	283,0 	58,99
100	1,043453		419,1

Stoffdaten von Wasser Quelle Wickipedia

Wasser hat unter Normaldruck seine größte Dichte von 1000 Kilogramm pro Kubikmeter bei 3,98 °C und zeigt damit eine Dichteanomalie. 
Diese besteht darin, dass sich Wasser unterhalb von 3,98 °C bei weiterer Temperaturverringerung, auch beim Wechsel zum festen 
Aggregatzustand, wieder ausdehnt, was man nur von wenigen Stoffen kennt. Die derzeit genauesten publizierten Werte für die maximale 
Dichte liegen bei (999,974950 ± 0,00084) kg/m³ und bei (3,983 ± 0,00067) °C für die Temperatur, bei der dieser Wert erreicht wird. 
Die Werte stellen einen Mittelwert der von verschiedenen physikalischen Instituten veröffentlichten Zahlen dar (Stand 2001).

Die Berechnung der Dichte von luftfreiem Wasser DLF in Abhängigkeit von der Temperatur T ([T] = °C) kann mit Hilfe der folgenden 
Virialgleichung erfolgen:
: \frac{D_{\rm LF}}{\rm g/l} = \frac{a_0 + a_1 T + a_2 T^2 + a_3 T^3 + a_4 T^4 + a_5 T^5}{1 + b T}.
mit den Koeffizienten: a0 = 999,83952; a1 = 16,952577 (°C)-1; a2 = -7,9905127·10-3 (°C)-2; a3 = -4,6241757·10-5 (°C)-3; 
a4 = 1,0584601·10-7 (°C)-4; a5 = -2,8103006·10-10 (°C)-5 und b = 0,0168872. 
Für die Berechnung der Dichte von luftgesättigtem Wasser korrigiert man den Wert nach 
DLG/(g/l) = DLF/(g/l) - 0,004612 + 0,000106 (°C)-1·T. (Quelle: PTB-Mitteilungen 100/3-90)

*)
END_FUNCTION

(* POU Building/HLK/WCT, ST *)
FUNCTION WCT : REAL
VAR_INPUT
	T : REAL;
	V : REAL;
END_VAR
VAR
END_VAR

(*
version 1.1	7 dec 2007
programmer 	hugo
tested by		tobias

this function calculates the wind chill temperature

*)
IF V < 5 OR T > 10 THEN
	WCT := T;
ELSE
	WCT := 13.12 + 0.6215 * T +(0.3965 * T - 11.37) * EXP(LN(v) * 0.16);
END_IF;


(* revision history
hm		7 feb 2007
	original version

hm		7 dec 2007
	changed code for better performance

*)
END_FUNCTION

(* POU Building/Jalousie/BLIND_ACTUATOR, ST *)
 FUNCTION_BLOCK BLIND_ACTUATOR
VAR_INPUT
	UP, DN : BOOL;
	S_IN : BYTE;
	T_UD : TIME := T#10s;
	T_ANGLE : TIME := T#3s;
END_VAR
VAR_INPUT CONSTANT
	T_LOCKOUT : TIME := t#100ms;
END_VAR
VAR_OUTPUT
	POS, ANG : BYTE;
	QU, QD : BOOL;
	STATUS : BYTE;
END_VAR
VAR
	position, angle : RMP_B;
	lock : INTERLOCK;
END_VAR

(*
version 1.2	18. oct. 2008
programmer 	hugo
tested by	oscat

blind actuator drives the up and down motor of a blind. T_lockout specifies the time between up or dn becomes active. 
To change direction there must be a minimum wait time to allow the motors to come to rest first.
the up and down outputs QU and QD are controlled by the inputs UP and DN.
the outputs pos and ang simulate the position of the blind pos = 0 means blind is down and pos = 255 = blind is up.
the angle 0 means vertical posisition of the slates and 255 means horizontal position of the slates.


*)
(* make sure only one motor is active at a given time *)
lock(i1 := UP, I2 := DN, TL := T_lockout);

(* ramp up or down to simulate the angle position of the blind slats *)
angle(e := lock.Q1 OR lock.Q2, UP := lock.Q1, PT := T_Angle);
position(e := lock.Q1 AND angle.high OR lock.Q2 AND angle.low, up := lock.Q1, PT := T_UD);

(* set the outputs *)
pos := position.Out;
ang := angle.Out;
QU := lock.Q1;
QD := lock.Q2;

(* set the status output *)
IF UP AND DN THEN
	IF s_in < 10 AND S_in > 1 THEN status := s_in; ELSE status := 1; END_IF;			(* error up and down together are not allowed *)
ELSIF S_IN > 0 THEN
	status := S_IN;
ELSIF UP THEN
	status := 101;
ELSIF DN THEN
	status := 102;
ELSE
	status := 0;
END_IF;


(* revision history
hm	29. sep 2007	rev 1.0
	original release

hm	6. oct 2007		rev 1.1
	rearanged outputs

hm	18. oct. 2008	rev 1.2
	changed calls for rmp_B because of change in RMP_B
*)
END_FUNCTION_BLOCK

(* POU Engineering/signal generators/RMP_B, ST *)
FUNCTION_BLOCK RMP_B
VAR_INPUT
	SET : BOOL;
	PT : TIME;
	E : BOOL := TRUE;
	UP : BOOL := TRUE;
	RST : BOOL;
END_VAR
VAR_OUTPUT
	OUT : BYTE;
	BUSY: BOOL;
	HIGH : BOOL;
	LOW : BOOL;
END_VAR
VAR
	rmp : _RMP_B;
END_VAR


(*
version 2.0	23. oct. 2008
programmer 	oscat
tested BY	oscat

this ramp generator generates a byte wide ramp with 255 steps
the generator has an asynchronous set and reset
the ramp is controlled by PT which is the total ramp time for a full sweep from 0..255
an UD input controlls the direction Up or Down and the E input enables the ramp generation
a busy output indicates that the ramp is running, busy false means output is stable.
the outputs low and high will be true when the output has reached its max or min value.

*)
(* generate ramp *)
rmp(dir := UP, E := E, TR := PT, rmp := out);

(* set or reset operation *)
IF RST THEN
	out := 0;
ELSIF SET THEN
	out := 255;
END_IF;

(* checks for outputs stable and reset or set busy flag *)
low := out = 0;
high := out = 255;
busy := NOT (low OR high) AND E;


(* revision history

hm 5.10.2006	rev 1.1
	added busy output
hm 17.1.2007	rev 1.2
	renamed input ud to up for better usability
	deleted unused variable step

hm	17.9.2007		rev 1.3
	replaced time() with t_plc_ms() for compatibility reasons

hm	28. sep 2007	rev 1.4
	added outputs on and off
	busy is now disabled while en is false
	new coding for higher accuracy and performance

hm	5. oct 2007	rev 1.5
	added statements to allow for PT to be t#0s output jumps to max or min immediately

hm	25. dec 2007	rev 1.6
	improved code for better performance

hm	16. oct. 2008	rev 1.7
	improved code for better performance

hm	18. oct. 2008	rev 1.8
	added type conversion to avoid warnings
	changed input en to e for compatibility reasons

hm	23. oct. 2008	REV 	2.0
	new code using _RMP_B

*)
END_FUNCTION_BLOCK

(* POU Engineering/automation/INTERLOCK, ST *)
FUNCTION_BLOCK INTERLOCK
VAR_INPUT
	I1, I2 : BOOL;
	TL : TIME;
END_VAR
VAR_OUTPUT
	Q1, Q2 : BOOL;
END_VAR
VAR
	T1, T2 : TOF;
END_VAR

(*
version 1.0	28 sep 2007
programmer 	hugo
tested by		tobias

INTERLOCK has two inputs I1 and I2 which drive the corresponding outputs Q1 and Q2.
the inputs signals lock each other out and therfore I1 can only drive Q1 when I2 is Low and vice versa.
The input TL specifies a dead time between two outputs can become active.
an output can only become active when the other output was not active for the time TL.

*)
(* the input signal have a run delay to lockout the other input *)
T1(IN := I1, PT := TL);
T2(IN := I2, PT := TL);

Q1 := I1 AND NOT t2.Q;
Q2 := I2 AND NOT t1.Q;


(* revision history

hm	28 sep 2007		rev 1.0
	original version

*)
END_FUNCTION_BLOCK

(* POU Building/Jalousie/BLIND_CONTROL, ST *)
FUNCTION_BLOCK BLIND_CONTROL
VAR_INPUT
	UP, DN : BOOL;
	S_IN : BYTE;
	PI : BYTE;
	AI : BYTE;
	T_UD, T_ANGLE : TIME;
END_VAR
VAR_INPUT CONSTANT
	SENS : BYTE := 5;
	T_LOCKOUT: TIME := T#100ms;
END_VAR
VAR_OUTPUT
	POS, ANG : BYTE;
	MU, MD : BOOL;
	STATUS : BYTE;
END_VAR
VAR
	act : BLIND_ACTUATOR;
	delta : BYTE;
END_VAR

(*
version 1.3	30. oct 2007
programmer 	hugo
tested by		tobias


*)
IF UP AND DN THEN
	(* automatic modus detected *)
	(* first find correct position *)
	IF BYTE_TO_INT(act.pos) < BYTE_TO_INT(pi) - delta THEN
		act.UP := TRUE;
		act.DN := FALSE;
		delta := 0;
		act.S_IN := 121;
	ELSIF BYTE_TO_INT(act.pos) > BYTE_TO_INT(pi) + delta THEN
		act.UP := FALSE;
		act.DN := TRUE;
		delta := 0;
		act.S_IN := 122;
	(* regulate angle *)
	ELSIF BYTE_TO_INT(act.ang) < BYTE_TO_INT(ai) - delta AND T_angle > T#100ms THEN
		act.UP := TRUE;
		act.DN := FALSE;
		delta := 0;
		act.S_IN := 123;
	ELSIF BYTE_TO_INT(act.ang) > BYTE_TO_INT(ai) + delta AND T_angle > T#100ms THEN
		act.UP := FALSE;
		act.DN := TRUE;
		delta := 0;
		act.S_IN := 124;
	(* correct position reached *)
	ELSE
		act.UP := FALSE;
		act.DN := FALSE;
		delta := sens;
		act.S_IN := 0;
	END_IF;
ELSE
	act.UP := UP;
	act.DN := DN;
END_IF;

(* hand over status *)
IF s_in > 0 THEN act.S_IN := S_IN; END_IF;

(* blind control calls blind_actuator *)
act(T_UD:=T_UD, T_ANGLE:=T_ANGLE, T_lockout := T_Lockout);
pos := act.pos;
ang := act.ang;
MU := act.QU;
md := act.QD;
status := act.status;

(* revision history
hm	29. sep 2007	rev 1.0
	original release

hm	6. oct 2007		rev 1.1
	rearranged outputs
	integrated blind_actuator into blind_control

hm	16. oct 2007	rev 1.2
	ignore angle when t_angle = 0

hm 29. oct 2007	rev 1.3
	added lockout configuration time for motor direction change
	sens has a setup value of 5
*)
END_FUNCTION_BLOCK

(* POU Building/Jalousie/BLIND_INPUT, ST *)
FUNCTION_BLOCK BLIND_INPUT
VAR_INPUT
	POS, ANG : BYTE;
	S1, S2 : BOOL;
	IN : BOOL;
	PI, AI : BYTE;
END_VAR
VAR_INPUT CONSTANT
	SINGLE_SWITCH : BOOL;
	CLICK_EN : BOOL := TRUE;
	CLICK_TIME : TIME := T#500ms;
	MAX_RUNTIME : TIME := T#60s;
	MANUAL_TIMEOUT: TIME := T#1h;
	DEBOUNCE_TIME : TIME := T#20ms;
	DBL_CLK1 : BOOL := FALSE;
	DBL_POS1 : BYTE;
	DBL_ANG1 : BYTE;
	DBL_CLK2 : BOOL := FALSE;
	DBL_POS2 : BYTE := 255;
	DBL_ANG2 : BYTE := 255;
	D1_TOGGLE : BOOL := TRUE;
	D2_TOGGLE : BOOL := TRUE;
END_VAR
VAR_OUTPUT
	QU, QD : BOOL;
	STATUS : BYTE;
	PO, AO : BYTE;
	D1, D2 : BOOL;
END_VAR
VAR
	s1e, s2e : TOF;
	s1d, s2d : CLICK_MODE;
	dir : BOOL;
	tx, last : TIME;
END_VAR

(*
version 1.5	22. jan. 2009
programmer 	hugo
tested by		oscat


*)
(* read system timer *)
tx := DWORD_TO_TIME(T_PLC_MS());

(* inputs S1 and S2 are debounced and then decoded for multiple clicks *)
s1e(in := S1, pt := DEBOUNCE_TIME);
s2e(in := S2, pt := DEBOUNCE_TIME);
s1d(in := (s1e.Q AND NOT SINGLE_SWITCH) OR (s1e.Q AND SINGLE_SWITCH AND dir), t_long := CLICK_TIME);
s2d(in := (s2e.Q AND NOT SINGLE_SWITCH) OR (s1e.Q AND SINGLE_SWITCH AND NOT dir), t_long := CLICK_TIME);

(* if d1 and d2 are not toggle clear them to make sure they are only active for oine cycle *)
IF NOT d1_toggle THEN d1 := FALSE; END_IF;
IF NOT d2_toggle THEN d2 := FALSE; END_IF;

(* decode actions *)
IF s1d.tp_LONG THEN
	status := 132;
ELSIF s2d.tp_LONG THEN
	status := 133;
ELSIF  s1d.SINGLE THEN
	IF click_en THEN
		(* if running then we stop otherwise start new direction *)
		IF QU XOR QD THEN
			status := 131;
		ELSE
			status := 134;
			last := tx;
			dir := NOT dir;
		END_IF;
	END_IF;
ELSIF  s2d.SINGLE THEN
	IF click_en THEN
		(* if running then we stop otherwise start new direction *)
		IF QU XOR QD THEN
			status := 131;
		ELSE
			status := 135;
			last := tx;
			dir := NOT dir;
		END_IF;
	END_IF;
ELSIF in THEN
	status := 136;
	last := tx;
ELSIF s1d.DOUBLE THEN
	IF dbl_clk1 THEN
		(* a position need to be set for a double click on S1 *)
		status := 137;
		last := tx;
	ELSE
		(* toggle the output when dbl_clk1 is not active *)
		D1 := NOT D1;
	END_IF;
ELSIF s2d.DOUBLE THEN
	IF dbl_clk2 THEN
		(* a position need to be set for a double click on S2 *)
		status := 138;
		last := tx;
	ELSE
		(* toggle the output when dbl_clk2 is not active *)
		(* in single switch mode we need to toggle d1 instead of d2 *)
		IF single_switch THEN D1 := NOT D1; ELSE D2 := NOT D2; END_IF;
	END_IF;
END_IF;


(* state machine *)
CASE status OF
	0:	(* automatic standby operation *)
			QU := QD := TRUE;
			PO := POS; AO := ANG;
	131:	(* manual operation standby *)
			QU := QD := FALSE;
			(* manual mode will be ended when timeout is reached *)
			IF tx - last >= manual_timeout THEN status := 0; END_IF;
	132:	(* manual operation up *)
			QU := TRUE; QD := FALSE;
			PO := POS; AO := ANG;
			last := tx;
			IF NOT s1d.LONG THEN status := 131; dir := NOT dir; END_IF;
	133:	(* manual operation down *)
			QU := FALSE; QD := TRUE;
			PO := POS; AO := ANG;
			last := tx;
			IF NOT s2d.LONG THEN	status := 131; dir := NOT dir; END_IF;
	134:	(* manual operation single click up *)
			QU := TRUE; QD := FALSE;
			PO := POS; AO := ANG;
			IF tx - last >= max_runtime THEN status := 131; END_IF;
	135:	(* manual operation single click dn *)
			QU := FALSE; QD := TRUE;
			PO := POS; AO := ANG;
			IF tx - last >= max_runtime THEN status := 131;	END_IF;
	136:	(* forced input in = true *)
			QU := QD := TRUE;
			PO := PI; AO := AI;
			IF tx-last >= max_runtime THEN status := 0; END_IF;
	137:	(* double click1 position *)
			QU := QD := TRUE;
			PO := DBL_POS1;
			AO := DBL_ANG1;
			IF tx - last >= max_runtime THEN status := 131; END_IF;
	138:	(* double click2 position *)
			QU := QD := TRUE;
			PO := DBL_POS2;
			AO := DBL_ANG2;
			IF tx - last >= max_runtime THEN status := 131; END_IF;
END_CASE




(* revision history
hm	29. sep 2007	rev 1.0
	original release

hm	6. oct 2007		rev 1.1
	renamed ps and as to po and ao

hm	30. dec 2007	rev 1.2
	added click_timeout variable and function

hm	16. jul. 2008	rev 1.3
	rewirtten code to allow for more functionality
	added single click mode with single_switch.
	added Debounce for inputs S1 and S2
	added double_click functionality

hm	26. sep. 2008	rev 1.4
	corrected an error while POS and ANG was transferred to outputs PO and AO during automatic modes

hm	22. jan 2009	rev 1.5
	added pulse mode for double click outputs
	added automatic mode for IN
*)
END_FUNCTION_BLOCK

(* POU Building/Jalousie/BLIND_NIGHT, ST *)
FUNCTION_BLOCK BLIND_NIGHT
VAR_INPUT
	UP, DN : BOOL;
	S_IN : BYTE;
	PI, AI : BYTE;
	E_NIGHT : BOOL := TRUE;
	E_DAY	: BOOL := TRUE;
	DTIN : DT;
	SUNRISE, SUNSET : TOD;
END_VAR
VAR_INPUT CONSTANT
	sunrise_offset : TIME;
	sunset_offset : TIME;
	night_position : BYTE;
	night_angle : BYTE;
END_VAR
VAR_OUTPUT
	QU, QD : BOOL;
	STATUS : BYTE;
	PO, AO : BYTE;
END_VAR
VAR
	night : BOOL;
	last_night, last_day : DATE;
END_VAR

(*
version 1.2	6 oct 2007
programmer 	hugo
tested by		tobias


*)
IF NOT (up AND dn) AND night THEN
	(* manual operation at night will cancel operation for one night *)
	night := FALSE;
ELSIF (DT_TO_TOD(dtin) > sunset + sunset_offset) AND (last_night < DT_TO_DATE(dtin)) AND NOT night AND e_night THEN
	(* enable night *)
	night := TRUE;
	last_night := DT_TO_DATE(dtin);
ELSIF (DT_TO_TOD(dtin) > sunrise + sunrise_offset) AND (last_day < DT_TO_DATE(dtin)) AND night AND e_day AND (last_night < DT_TO_DATE(dtin)) THEN
	(* disable night *)
	night := FALSE;
	last_day := DT_TO_DATE(dtin);
END_IF;

(* shade at night only in auto mode and enable = true *)
IF UP AND DN AND night THEN
	status := 141;
	po := night_position;
	ao := night_angle;
ELSE
	QU := UP;
	QD := DN;
	po := pi;
	ao := ai;
	status := s_in;
END_IF;


(* revision history
hm	29. sep 2007	rev 1.0
	original version

hm	5. oct 2007		rev 1.1
	added enable input

hm	6. oct 2007		rev 1.2
	added pos and angle inputs and outputs
	night position and angle can now be configured
	any manual operation at night will cancel night operation

